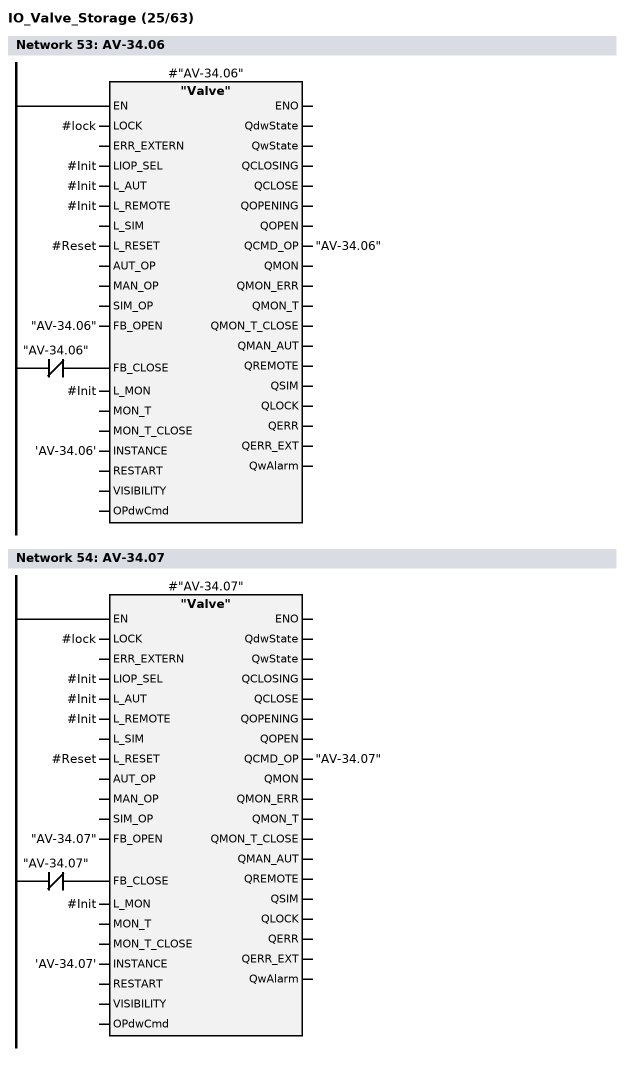
   RUNG wire#powerrail
      #"AV-34.06"(FB_CLOSE := wire#w1, LOCK := #lock, ERR_EXTERN :=, LIOP_SEL := #Init, L_AUT := #Init, L_REMOTE := #Init, L_SIM :=, L_RESET := #Reset, AUT_OP :=, MAN_OP :=, SIM_OP :=, FB_OPEN := "AV-34.06", L_MON := #Init, MON_T :=, MON_T_CLOSE :=, INSTANCE := 'AV-34.06', RESTART :=, VISIBILITY :=, OPdwCmd :=, QdwState =>, QwState =>, QCLOSING =>, QCLOSE =>, QOPENING =>, QOPEN =>, QCMD_OP => "AV-34.06", QMON =>, QMON_ERR =>, QMON_T =>, QMON_T_CLOSE =>, QMAN_AUT =>, QREMOTE =>, QSIM =>, QLOCK =>, QERR =>, QERR_EXT =>, QwAlarm =>)
   END_RUNG
   RUNG wire#powerrail
      I_Contact( "AV-34.06" )
   END_RUNG wire#w1
   // the same network as SCL:
   #"AV-34.06"(LOCK := #lock,   // "Valve"
               LIOP_SEL := #Init,
               L_AUT := #Init,
               L_REMOTE := #Init,
               L_RESET := #Reset,
               FB_OPEN := "AV-34.06",
               FB_CLOSE := NOT "AV-34.06",
               L_MON := #Init,
               INSTANCE := 'AV-34.06',
               QCMD_OP => "AV-34.06");
END_REGION

REGION Network 54: AV-34.07
   RUNG wire#powerrail
      #"AV-34.07"(FB_CLOSE := wire#w1, LOCK := #lock, ERR_EXTERN :=, LIOP_SEL := #Init, L_AUT := #Init, L_REMOTE := #Init, L_SIM :=, L_RESET := #Reset, AUT_OP :=, MAN_OP :=, SIM_OP :=, FB_OPEN := "AV-34.07", L_MON := #Init, MON_T :=, MON_T_CLOSE :=, INSTANCE := 'AV-34.07', RESTART :=, VISIBILITY :=, OPdwCmd :=, QdwState =>, QwState =>, QCLOSING =>, QCLOSE =>, QOPENING =>, QOPEN =>, QCMD_OP => "AV-34.07", QMON =>, QMON_ERR =>, QMON_T =>, QMON_T_CLOSE =>, QMAN_AUT =>, QREMOTE =>, QSIM =>, QLOCK =>, QERR =>, QERR_EXT =>, QwAlarm =>)
   END_RUNG
   RUNG wire#powerrail
      I_Contact( "AV-34.07" )
   END_RUNG wire#w1
   // the same network as SCL:
   #"AV-34.07"(LOCK := #lock,   // "Valve"
               LIOP_SEL := #Init,
               L_AUT := #Init,
               L_REMOTE := #Init,
               L_RESET := #Reset,
               FB_OPEN := "AV-34.07",
               FB_CLOSE := NOT "AV-34.07",
               L_MON := #Init,
               INSTANCE := 'AV-34.07',
               QCMD_OP => "AV-34.07");
END_REGION

REGION Network 55: AV-34.08
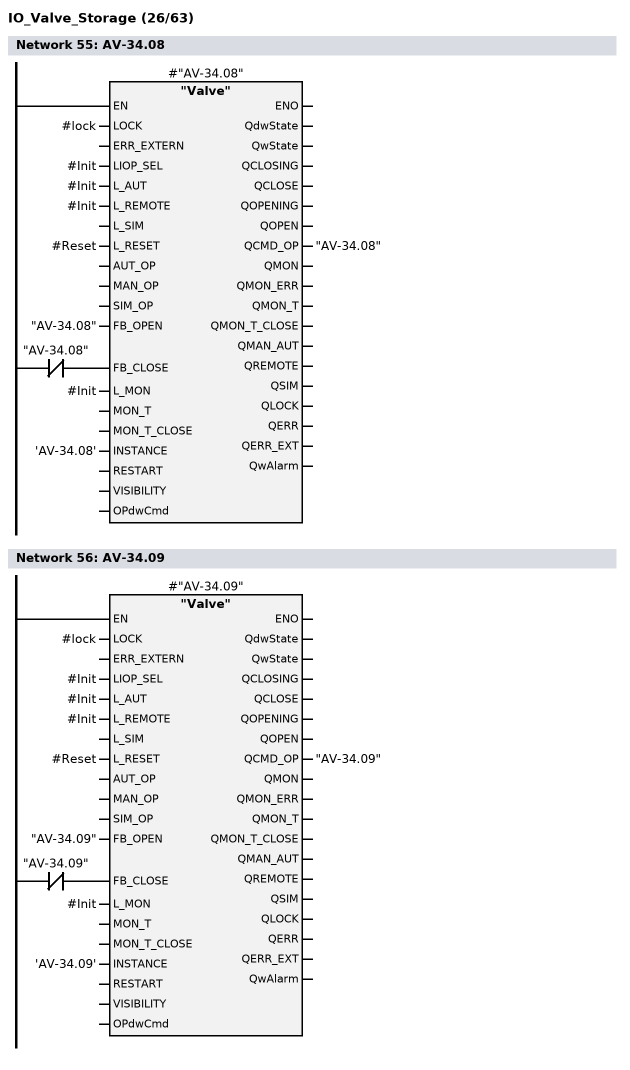
   RUNG wire#powerrail
      #"AV-34.08"(FB_CLOSE := wire#w1, LOCK := #lock, ERR_EXTERN :=, LIOP_SEL := #Init, L_AUT := #Init, L_REMOTE := #Init, L_SIM :=, L_RESET := #Reset, AUT_OP :=, MAN_OP :=, SIM_OP :=, FB_OPEN := "AV-34.08", L_MON := #Init, MON_T :=, MON_T_CLOSE :=, INSTANCE := 'AV-34.08', RESTART :=, VISIBILITY :=, OPdwCmd :=, QdwState =>, QwState =>, QCLOSING =>, QCLOSE =>, QOPENING =>, QOPEN =>, QCMD_OP => "AV-34.08", QMON =>, QMON_ERR =>, QMON_T =>, QMON_T_CLOSE =>, QMAN_AUT =>, QREMOTE =>, QSIM =>, QLOCK =>, QERR =>, QERR_EXT =>, QwAlarm =>)
   END_RUNG
   RUNG wire#powerrail
      I_Contact( "AV-34.08" )
   END_RUNG wire#w1
   // the same network as SCL:
   #"AV-34.08"(LOCK := #lock,   // "Valve"
               LIOP_SEL := #Init,
               L_AUT := #Init,
               L_REMOTE := #Init,
               L_RESET := #Reset,
               FB_OPEN := "AV-34.08",
               FB_CLOSE := NOT "AV-34.08",
               L_MON := #Init,
               INSTANCE := 'AV-34.08',
               QCMD_OP => "AV-34.08");
END_REGION

REGION Network 56: AV-34.09
   RUNG wire#powerrail
      #"AV-34.09"(FB_CLOSE := wire#w1, LOCK := #lock, ERR_EXTERN :=, LIOP_SEL := #Init, L_AUT := #Init, L_REMOTE := #Init, L_SIM :=, L_RESET := #Reset, AUT_OP :=, MAN_OP :=, SIM_OP :=, FB_OPEN := "AV-34.09", L_MON := #Init, MON_T :=, MON_T_CLOSE :=, INSTANCE := 'AV-34.09', RESTART :=, VISIBILITY :=, OPdwCmd :=, QdwState =>, QwState =>, QCLOSING =>, QCLOSE =>, QOPENING =>, QOPEN =>, QCMD_OP => "AV-34.09", QMON =>, QMON_ERR =>, QMON_T =>, QMON_T_CLOSE =>, QMAN_AUT =>, QREMOTE =>, QSIM =>, QLOCK =>, QERR =>, QERR_EXT =>, QwAlarm =>)
   END_RUNG
   RUNG wire#powerrail
      I_Contact( "AV-34.09" )
   END_RUNG wire#w1
   // the same network as SCL:
   #"AV-34.09"(LOCK := #lock,   // "Valve"
               LIOP_SEL := #Init,
               L_AUT := #Init,
               L_REMOTE := #Init,
               L_RESET := #Reset,
               FB_OPEN := "AV-34.09",
               FB_CLOSE := NOT "AV-34.09",
               L_MON := #Init,
               INSTANCE := 'AV-34.09',
               QCMD_OP => "AV-34.09");
END_REGION

REGION Network 57: AV-34.10
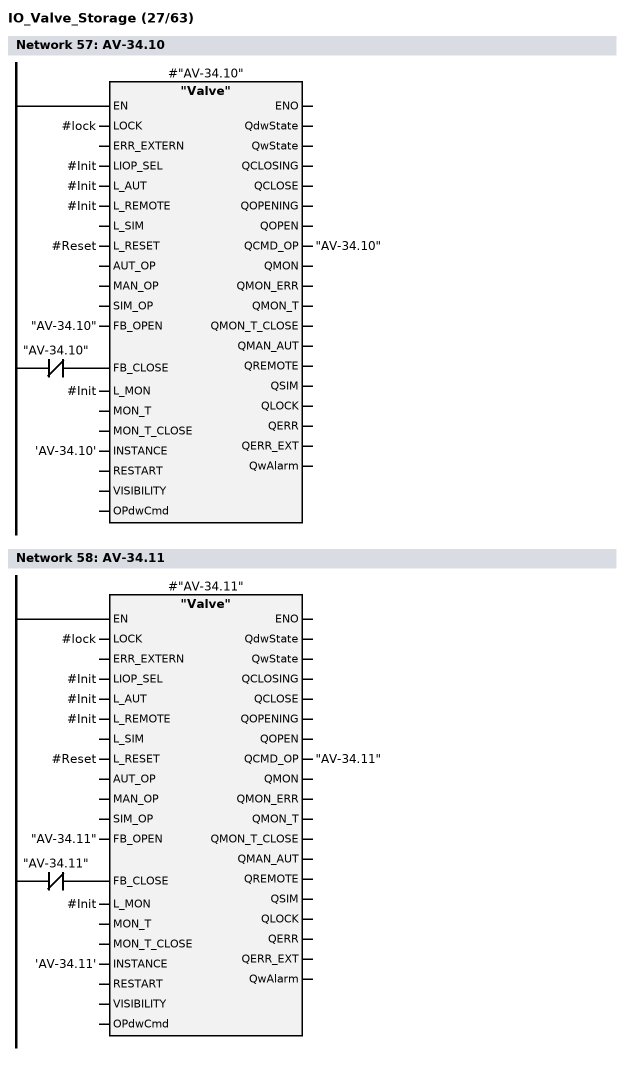
   RUNG wire#powerrail
      #"AV-34.10"(FB_CLOSE := wire#w1, LOCK := #lock, ERR_EXTERN :=, LIOP_SEL := #Init, L_AUT := #Init, L_REMOTE := #Init, L_SIM :=, L_RESET := #Reset, AUT_OP :=, MAN_OP :=, SIM_OP :=, FB_OPEN := "AV-34.10", L_MON := #Init, MON_T :=, MON_T_CLOSE :=, INSTANCE := 'AV-34.10', RESTART :=, VISIBILITY :=, OPdwCmd :=, QdwState =>, QwState =>, QCLOSING =>, QCLOSE =>, QOPENING =>, QOPEN =>, QCMD_OP => "AV-34.10", QMON =>, QMON_ERR =>, QMON_T =>, QMON_T_CLOSE =>, QMAN_AUT =>, QREMOTE =>, QSIM =>, QLOCK =>, QERR =>, QERR_EXT =>, QwAlarm =>)
   END_RUNG
   RUNG wire#powerrail
      I_Contact( "AV-34.10" )
   END_RUNG wire#w1
   // the same network as SCL:
   #"AV-34.10"(LOCK := #lock,   // "Valve"
               LIOP_SEL := #Init,
               L_AUT := #Init,
               L_REMOTE := #Init,
               L_RESET := #Reset,
               FB_OPEN := "AV-34.10",
               FB_CLOSE := NOT "AV-34.10",
               L_MON := #Init,
               INSTANCE := 'AV-34.10',
               QCMD_OP => "AV-34.10");
END_REGION

REGION Network 58: AV-34.11
   RUNG wire#powerrail
      #"AV-34.11"(FB_CLOSE := wire#w1, LOCK := #lock, ERR_EXTERN :=, LIOP_SEL := #Init, L_AUT := #Init, L_REMOTE := #Init, L_SIM :=, L_RESET := #Reset, AUT_OP :=, MAN_OP :=, SIM_OP :=, FB_OPEN := "AV-34.11", L_MON := #Init, MON_T :=, MON_T_CLOSE :=, INSTANCE := 'AV-34.11', RESTART :=, VISIBILITY :=, OPdwCmd :=, QdwState =>, QwState =>, QCLOSING =>, QCLOSE =>, QOPENING =>, QOPEN =>, QCMD_OP => "AV-34.11", QMON =>, QMON_ERR =>, QMON_T =>, QMON_T_CLOSE =>, QMAN_AUT =>, QREMOTE =>, QSIM =>, QLOCK =>, QERR =>, QERR_EXT =>, QwAlarm =>)
   END_RUNG
   RUNG wire#powerrail
      I_Contact( "AV-34.11" )
   END_RUNG wire#w1
   // the same network as SCL:
   #"AV-34.11"(LOCK := #lock,   // "Valve"
               LIOP_SEL := #Init,
               L_AUT := #Init,
               L_REMOTE := #Init,
               L_RESET := #Reset,
               FB_OPEN := "AV-34.11",
               FB_CLOSE := NOT "AV-34.11",
               L_MON := #Init,
               INSTANCE := 'AV-34.11',
               QCMD_OP => "AV-34.11");
END_REGION

REGION Network 59: AV-34.12
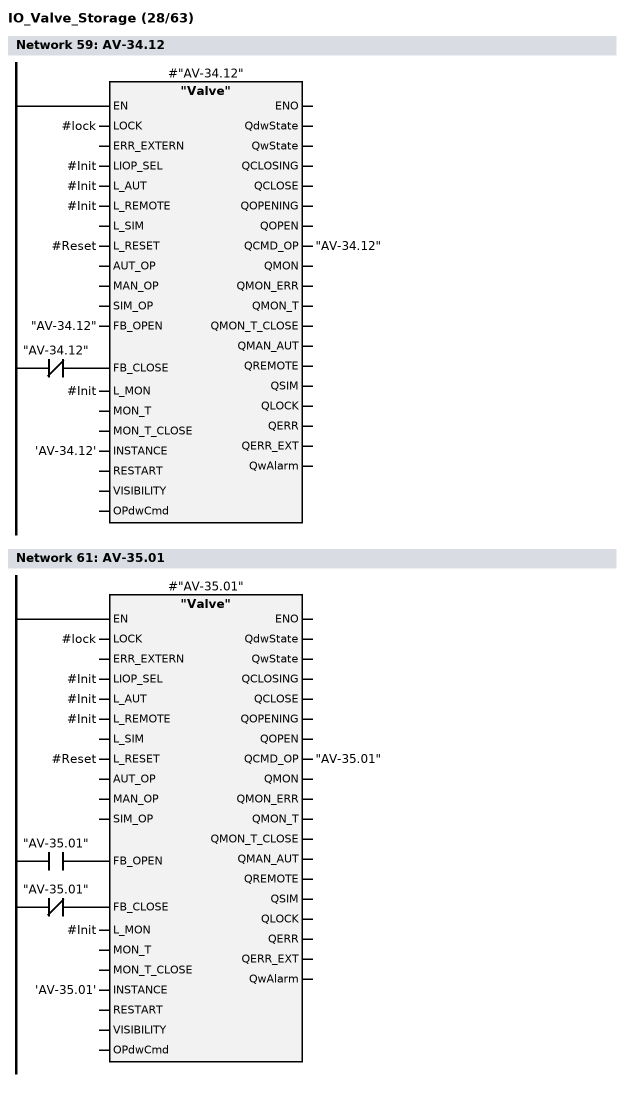
   RUNG wire#powerrail
      #"AV-34.12"(FB_CLOSE := wire#w1, LOCK := #lock, ERR_EXTERN :=, LIOP_SEL := #Init, L_AUT := #Init, L_REMOTE := #Init, L_SIM :=, L_RESET := #Reset, AUT_OP :=, MAN_OP :=, SIM_OP :=, FB_OPEN := "AV-34.12", L_MON := #Init, MON_T :=, MON_T_CLOSE :=, INSTANCE := 'AV-34.12', RESTART :=, VISIBILITY :=, OPdwCmd :=, QdwState =>, QwState =>, QCLOSING =>, QCLOSE =>, QOPENING =>, QOPEN =>, QCMD_OP => "AV-34.12", QMON =>, QMON_ERR =>, QMON_T =>, QMON_T_CLOSE =>, QMAN_AUT =>, QREMOTE =>, QSIM =>, QLOCK =>, QERR =>, QERR_EXT =>, QwAlarm =>)
   END_RUNG
   RUNG wire#powerrail
      I_Contact( "AV-34.12" )
   END_RUNG wire#w1
   // the same network as SCL:
   #"AV-34.12"(LOCK := #lock,   // "Valve"
               LIOP_SEL := #Init,
               L_AUT := #Init,
               L_REMOTE := #Init,
               L_RESET := #Reset,
               FB_OPEN := "AV-34.12",
               FB_CLOSE := NOT "AV-34.12",
               L_MON := #Init,
               INSTANCE := 'AV-34.12',
               QCMD_OP => "AV-34.12");
END_REGION

REGION Network 61: AV-35.01
   RUNG wire#powerrail
      #"AV-35.01"(FB_OPEN := wire#w1, FB_CLOSE := wire#w2, LOCK := #lock, ERR_EXTERN :=, LIOP_SEL := #Init, L_AUT := #Init, L_REMOTE := #Init, L_SIM :=, L_RESET := #Reset, AUT_OP :=, MAN_OP :=, SIM_OP :=, L_MON := #Init, MON_T :=, MON_T_CLOSE :=, INSTANCE := 'AV-35.01', RESTART :=, VISIBILITY :=, OPdwCmd :=, QdwState =>, QwState =>, QCLOSING =>, QCLOSE =>, QOPENING =>, QOPEN =>, QCMD_OP => "AV-35.01", QMON =>, QMON_ERR =>, QMON_T =>, QMON_T_CLOSE =>, QMAN_AUT =>, QREMOTE =>, QSIM =>, QLOCK =>, QERR =>, QERR_EXT =>, QwAlarm =>)
   END_RUNG
   RUNG wire#powerrail
      Contact( "AV-35.01" )
   END_RUNG wire#w1
   RUNG wire#powerrail
      I_Contact( "AV-35.01" )
   END_RUNG wire#w2
   // the same network as SCL:
   #"AV-35.01"(LOCK := #lock,   // "Valve"
               LIOP_SEL := #Init,
               L_AUT := #Init,
               L_REMOTE := #Init,
               L_RESET := #Reset,
               FB_OPEN := "AV-35.01",
               FB_CLOSE := NOT "AV-35.01",
               L_MON := #Init,
               INSTANCE := 'AV-35.01',
               QCMD_OP => "AV-35.01");
END_REGION

REGION Network 62: AV-35.02
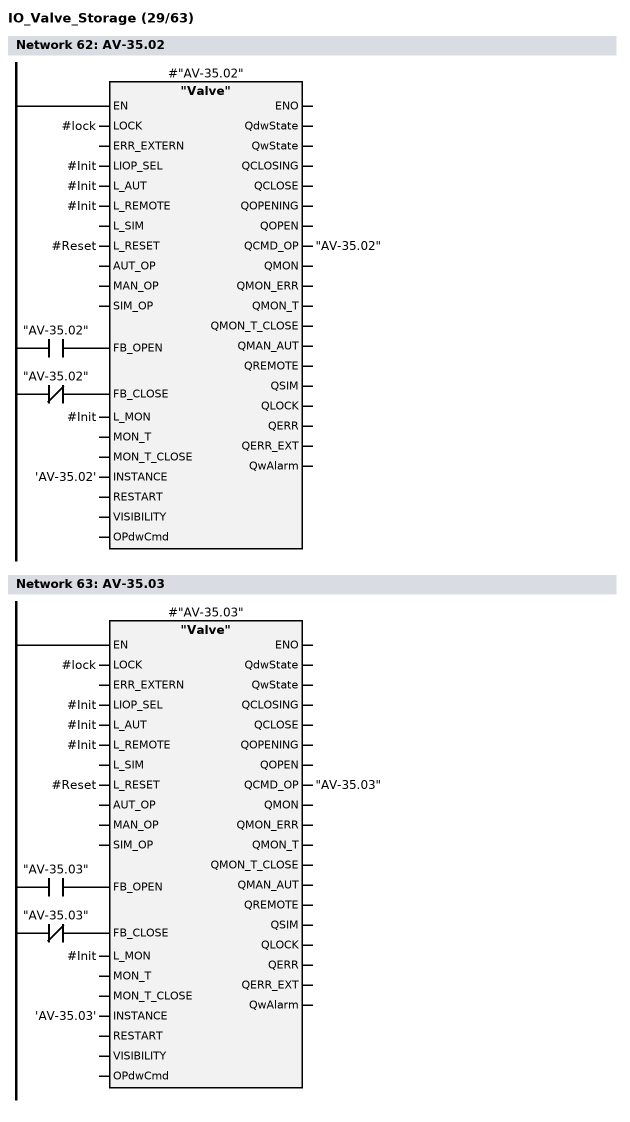
   RUNG wire#powerrail
      #"AV-35.02"(FB_OPEN := wire#w1, FB_CLOSE := wire#w2, LOCK := #lock, ERR_EXTERN :=, LIOP_SEL := #Init, L_AUT := #Init, L_REMOTE := #Init, L_SIM :=, L_RESET := #Reset, AUT_OP :=, MAN_OP :=, SIM_OP :=, L_MON := #Init, MON_T :=, MON_T_CLOSE :=, INSTANCE := 'AV-35.02', RESTART :=, VISIBILITY :=, OPdwCmd :=, QdwState =>, QwState =>, QCLOSING =>, QCLOSE =>, QOPENING =>, QOPEN =>, QCMD_OP => "AV-35.02", QMON =>, QMON_ERR =>, QMON_T =>, QMON_T_CLOSE =>, QMAN_AUT =>, QREMOTE =>, QSIM =>, QLOCK =>, QERR =>, QERR_EXT =>, QwAlarm =>)
   END_RUNG
   RUNG wire#powerrail
      Contact( "AV-35.02" )
   END_RUNG wire#w1
   RUNG wire#powerrail
      I_Contact( "AV-35.02" )
   END_RUNG wire#w2
   // the same network as SCL:
   #"AV-35.02"(LOCK := #lock,   // "Valve"
               LIOP_SEL := #Init,
               L_AUT := #Init,
               L_REMOTE := #Init,
               L_RESET := #Reset,
               FB_OPEN := "AV-35.02",
               FB_CLOSE := NOT "AV-35.02",
               L_MON := #Init,
               INSTANCE := 'AV-35.02',
               QCMD_OP => "AV-35.02");
END_REGION

REGION Network 63: AV-35.03
   RUNG wire#powerrail
      #"AV-35.03"(FB_OPEN := wire#w1, FB_CLOSE := wire#w2, LOCK := #lock, ERR_EXTERN :=, LIOP_SEL := #Init, L_AUT := #Init, L_REMOTE := #Init, L_SIM :=, L_RESET := #Reset, AUT_OP :=, MAN_OP :=, SIM_OP :=, L_MON := #Init, MON_T :=, MON_T_CLOSE :=, INSTANCE := 'AV-35.03', RESTART :=, VISIBILITY :=, OPdwCmd :=, QdwState =>, QwState =>, QCLOSING =>, QCLOSE =>, QOPENING =>, QOPEN =>, QCMD_OP => "AV-35.03", QMON =>, QMON_ERR =>, QMON_T =>, QMON_T_CLOSE =>, QMAN_AUT =>, QREMOTE =>, QSIM =>, QLOCK =>, QERR =>, QERR_EXT =>, QwAlarm =>)
   END_RUNG
   RUNG wire#powerrail
      Contact( "AV-35.03" )
   END_RUNG wire#w1
   RUNG wire#powerrail
      I_Contact( "AV-35.03" )
   END_RUNG wire#w2
   // the same network as SCL:
   #"AV-35.03"(LOCK := #lock,   // "Valve"
               LIOP_SEL := #Init,
               L_AUT := #Init,
               L_REMOTE := #Init,
               L_RESET := #Reset,
               FB_OPEN := "AV-35.03",
               FB_CLOSE := NOT "AV-35.03",
               L_MON := #Init,
               INSTANCE := 'AV-35.03',
               QCMD_OP => "AV-35.03");
END_REGION

REGION Network 64: AV-35.04
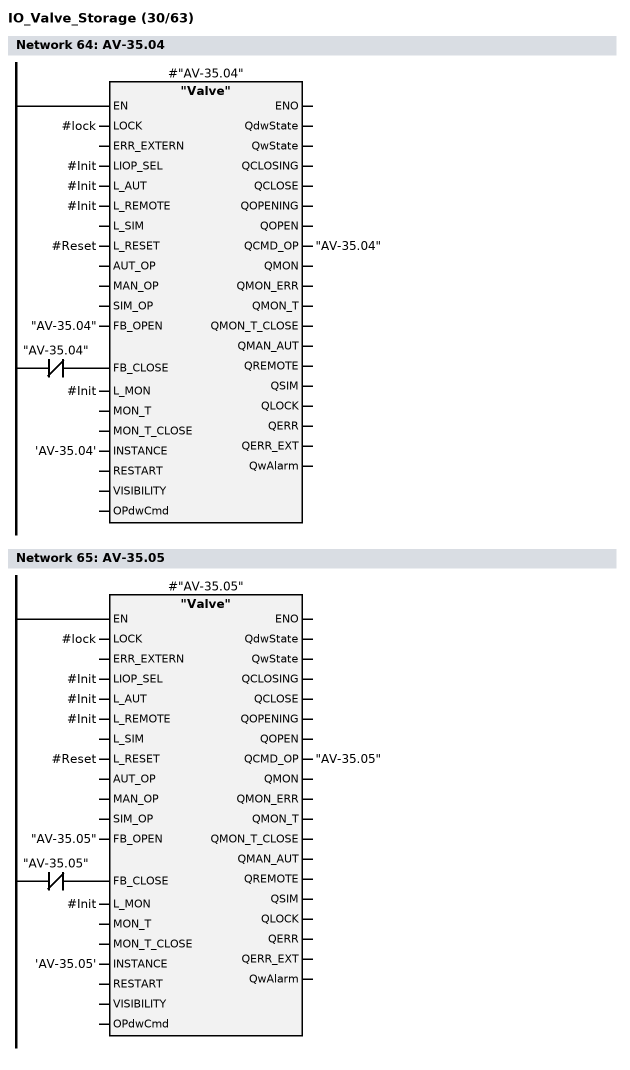
   RUNG wire#powerrail
      #"AV-35.04"(FB_CLOSE := wire#w1, LOCK := #lock, ERR_EXTERN :=, LIOP_SEL := #Init, L_AUT := #Init, L_REMOTE := #Init, L_SIM :=, L_RESET := #Reset, AUT_OP :=, MAN_OP :=, SIM_OP :=, FB_OPEN := "AV-35.04", L_MON := #Init, MON_T :=, MON_T_CLOSE :=, INSTANCE := 'AV-35.04', RESTART :=, VISIBILITY :=, OPdwCmd :=, QdwState =>, QwState =>, QCLOSING =>, QCLOSE =>, QOPENING =>, QOPEN =>, QCMD_OP => "AV-35.04", QMON =>, QMON_ERR =>, QMON_T =>, QMON_T_CLOSE =>, QMAN_AUT =>, QREMOTE =>, QSIM =>, QLOCK =>, QERR =>, QERR_EXT =>, QwAlarm =>)
   END_RUNG
   RUNG wire#powerrail
      I_Contact( "AV-35.04" )
   END_RUNG wire#w1
   // the same network as SCL:
   #"AV-35.04"(LOCK := #lock,   // "Valve"
               LIOP_SEL := #Init,
               L_AUT := #Init,
               L_REMOTE := #Init,
               L_RESET := #Reset,
               FB_OPEN := "AV-35.04",
               FB_CLOSE := NOT "AV-35.04",
               L_MON := #Init,
               INSTANCE := 'AV-35.04',
               QCMD_OP => "AV-35.04");
END_REGION

REGION Network 65: AV-35.05
   RUNG wire#powerrail
      #"AV-35.05"(FB_CLOSE := wire#w1, LOCK := #lock, ERR_EXTERN :=, LIOP_SEL := #Init, L_AUT := #Init, L_REMOTE := #Init, L_SIM :=, L_RESET := #Reset, AUT_OP :=, MAN_OP :=, SIM_OP :=, FB_OPEN := "AV-35.05", L_MON := #Init, MON_T :=, MON_T_CLOSE :=, INSTANCE := 'AV-35.05', RESTART :=, VISIBILITY :=, OPdwCmd :=, QdwState =>, QwState =>, QCLOSING =>, QCLOSE =>, QOPENING =>, QOPEN =>, QCMD_OP => "AV-35.05", QMON =>, QMON_ERR =>, QMON_T =>, QMON_T_CLOSE =>, QMAN_AUT =>, QREMOTE =>, QSIM =>, QLOCK =>, QERR =>, QERR_EXT =>, QwAlarm =>)
   END_RUNG
   RUNG wire#powerrail
      I_Contact( "AV-35.05" )
   END_RUNG wire#w1
   // the same network as SCL:
   #"AV-35.05"(LOCK := #lock,   // "Valve"
               LIOP_SEL := #Init,
               L_AUT := #Init,
               L_REMOTE := #Init,
               L_RESET := #Reset,
               FB_OPEN := "AV-35.05",
               FB_CLOSE := NOT "AV-35.05",
               L_MON := #Init,
               INSTANCE := 'AV-35.05',
               QCMD_OP => "AV-35.05");
END_REGION

REGION Network 66: AV-35.06
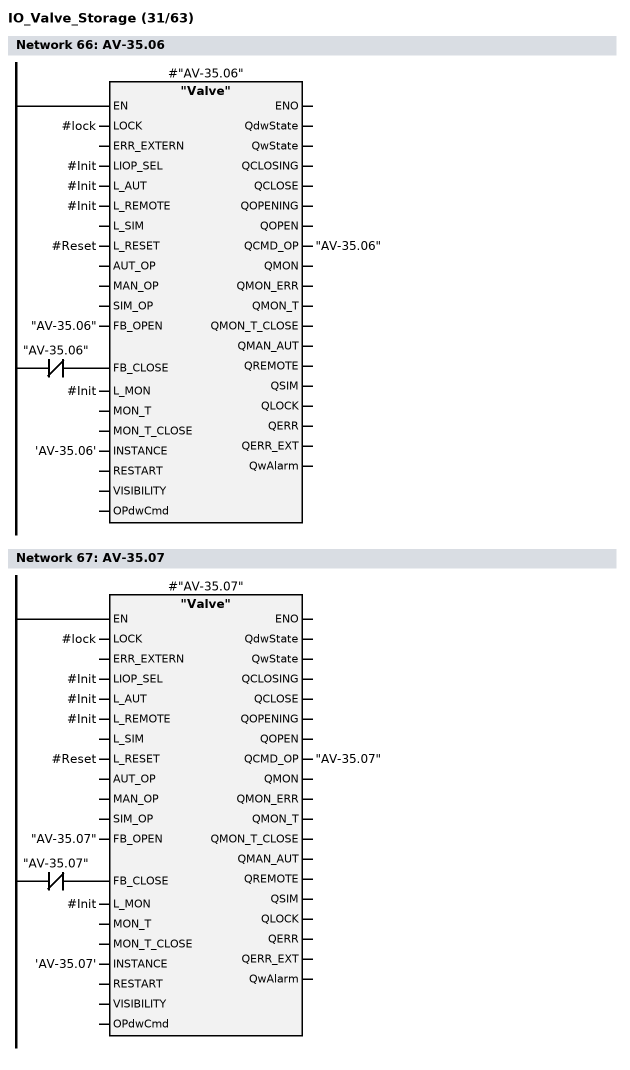
   RUNG wire#powerrail
      #"AV-35.06"(FB_CLOSE := wire#w1, LOCK := #lock, ERR_EXTERN :=, LIOP_SEL := #Init, L_AUT := #Init, L_REMOTE := #Init, L_SIM :=, L_RESET := #Reset, AUT_OP :=, MAN_OP :=, SIM_OP :=, FB_OPEN := "AV-35.06", L_MON := #Init, MON_T :=, MON_T_CLOSE :=, INSTANCE := 'AV-35.06', RESTART :=, VISIBILITY :=, OPdwCmd :=, QdwState =>, QwState =>, QCLOSING =>, QCLOSE =>, QOPENING =>, QOPEN =>, QCMD_OP => "AV-35.06", QMON =>, QMON_ERR =>, QMON_T =>, QMON_T_CLOSE =>, QMAN_AUT =>, QREMOTE =>, QSIM =>, QLOCK =>, QERR =>, QERR_EXT =>, QwAlarm =>)
   END_RUNG
   RUNG wire#powerrail
      I_Contact( "AV-35.06" )
   END_RUNG wire#w1
   // the same network as SCL:
   #"AV-35.06"(LOCK := #lock,   // "Valve"
               LIOP_SEL := #Init,
               L_AUT := #Init,
               L_REMOTE := #Init,
               L_RESET := #Reset,
               FB_OPEN := "AV-35.06",
               FB_CLOSE := NOT "AV-35.06",
               L_MON := #Init,
               INSTANCE := 'AV-35.06',
               QCMD_OP => "AV-35.06");
END_REGION

REGION Network 67: AV-35.07
   RUNG wire#powerrail
      #"AV-35.07"(FB_CLOSE := wire#w1, LOCK := #lock, ERR_EXTERN :=, LIOP_SEL := #Init, L_AUT := #Init, L_REMOTE := #Init, L_SIM :=, L_RESET := #Reset, AUT_OP :=, MAN_OP :=, SIM_OP :=, FB_OPEN := "AV-35.07", L_MON := #Init, MON_T :=, MON_T_CLOSE :=, INSTANCE := 'AV-35.07', RESTART :=, VISIBILITY :=, OPdwCmd :=, QdwState =>, QwState =>, QCLOSING =>, QCLOSE =>, QOPENING =>, QOPEN =>, QCMD_OP => "AV-35.07", QMON =>, QMON_ERR =>, QMON_T =>, QMON_T_CLOSE =>, QMAN_AUT =>, QREMOTE =>, QSIM =>, QLOCK =>, QERR =>, QERR_EXT =>, QwAlarm =>)
   END_RUNG
   RUNG wire#powerrail
      I_Contact( "AV-35.07" )
   END_RUNG wire#w1
   // the same network as SCL:
   #"AV-35.07"(LOCK := #lock,   // "Valve"
               LIOP_SEL := #Init,
               L_AUT := #Init,
               L_REMOTE := #Init,
               L_RESET := #Reset,
               FB_OPEN := "AV-35.07",
               FB_CLOSE := NOT "AV-35.07",
               L_MON := #Init,
               INSTANCE := 'AV-35.07',
               QCMD_OP => "AV-35.07");
END_REGION

REGION Network 68: AV-35.08
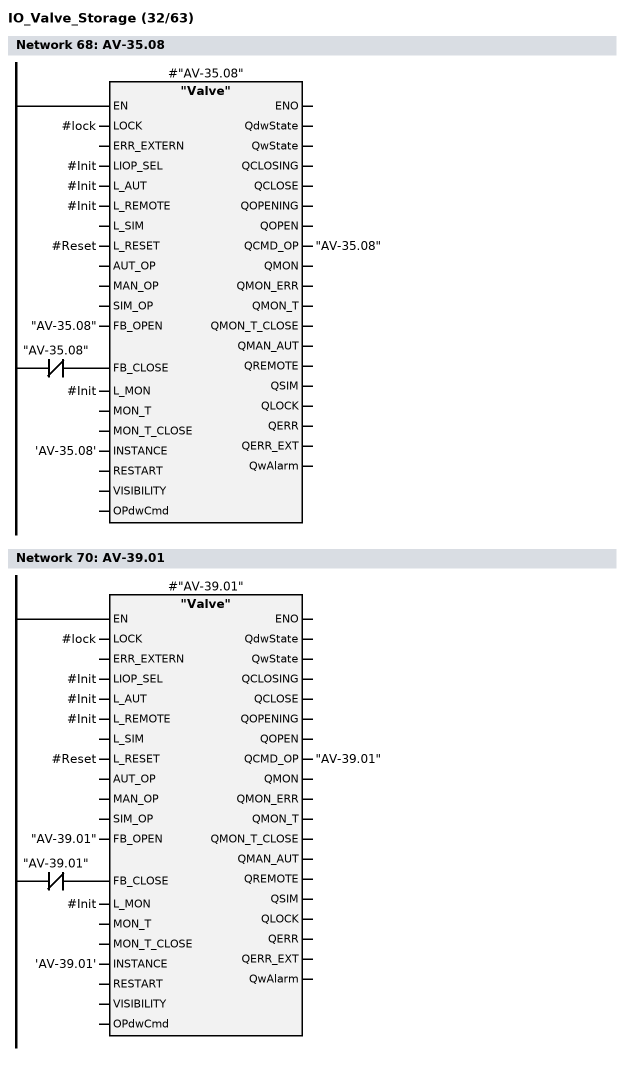
   RUNG wire#powerrail
      #"AV-35.08"(FB_CLOSE := wire#w1, LOCK := #lock, ERR_EXTERN :=, LIOP_SEL := #Init, L_AUT := #Init, L_REMOTE := #Init, L_SIM :=, L_RESET := #Reset, AUT_OP :=, MAN_OP :=, SIM_OP :=, FB_OPEN := "AV-35.08", L_MON := #Init, MON_T :=, MON_T_CLOSE :=, INSTANCE := 'AV-35.08', RESTART :=, VISIBILITY :=, OPdwCmd :=, QdwState =>, QwState =>, QCLOSING =>, QCLOSE =>, QOPENING =>, QOPEN =>, QCMD_OP => "AV-35.08", QMON =>, QMON_ERR =>, QMON_T =>, QMON_T_CLOSE =>, QMAN_AUT =>, QREMOTE =>, QSIM =>, QLOCK =>, QERR =>, QERR_EXT =>, QwAlarm =>)
   END_RUNG
   RUNG wire#powerrail
      I_Contact( "AV-35.08" )
   END_RUNG wire#w1
   // the same network as SCL:
   #"AV-35.08"(LOCK := #lock,   // "Valve"
               LIOP_SEL := #Init,
               L_AUT := #Init,
               L_REMOTE := #Init,
               L_RESET := #Reset,
               FB_OPEN := "AV-35.08",
               FB_CLOSE := NOT "AV-35.08",
               L_MON := #Init,
               INSTANCE := 'AV-35.08',
               QCMD_OP => "AV-35.08");
END_REGION

REGION Network 70: AV-39.01
   RUNG wire#powerrail
      #"AV-39.01"(FB_CLOSE := wire#w1, LOCK := #lock, ERR_EXTERN :=, LIOP_SEL := #Init, L_AUT := #Init, L_REMOTE := #Init, L_SIM :=, L_RESET := #Reset, AUT_OP :=, MAN_OP :=, SIM_OP :=, FB_OPEN := "AV-39.01", L_MON := #Init, MON_T :=, MON_T_CLOSE :=, INSTANCE := 'AV-39.01', RESTART :=, VISIBILITY :=, OPdwCmd :=, QdwState =>, QwState =>, QCLOSING =>, QCLOSE =>, QOPENING =>, QOPEN =>, QCMD_OP => "AV-39.01", QMON =>, QMON_ERR =>, QMON_T =>, QMON_T_CLOSE =>, QMAN_AUT =>, QREMOTE =>, QSIM =>, QLOCK =>, QERR =>, QERR_EXT =>, QwAlarm =>)
   END_RUNG
   RUNG wire#powerrail
      I_Contact( "AV-39.01" )
   END_RUNG wire#w1
   // the same network as SCL:
   #"AV-39.01"(LOCK := #lock,   // "Valve"
               LIOP_SEL := #Init,
               L_AUT := #Init,
               L_REMOTE := #Init,
               L_RESET := #Reset,
               FB_OPEN := "AV-39.01",
               FB_CLOSE := NOT "AV-39.01",
               L_MON := #Init,
               INSTANCE := 'AV-39.01',
               QCMD_OP => "AV-39.01");
END_REGION

REGION Network 71: AV-39.02
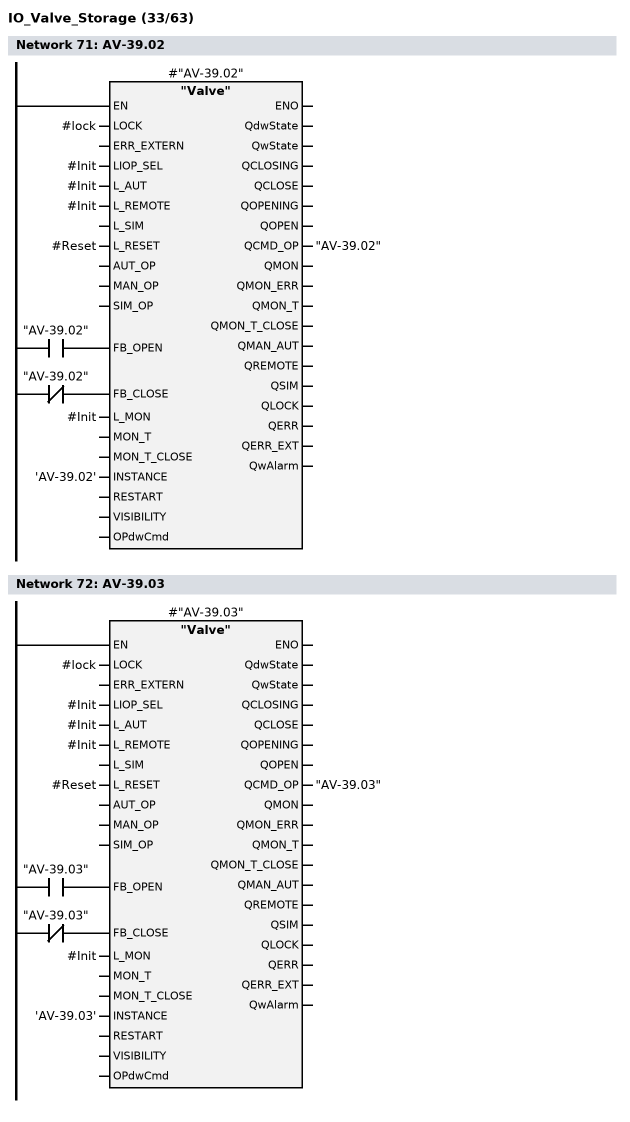
   RUNG wire#powerrail
      #"AV-39.02"(FB_OPEN := wire#w1, FB_CLOSE := wire#w2, LOCK := #lock, ERR_EXTERN :=, LIOP_SEL := #Init, L_AUT := #Init, L_REMOTE := #Init, L_SIM :=, L_RESET := #Reset, AUT_OP :=, MAN_OP :=, SIM_OP :=, L_MON := #Init, MON_T :=, MON_T_CLOSE :=, INSTANCE := 'AV-39.02', RESTART :=, VISIBILITY :=, OPdwCmd :=, QdwState =>, QwState =>, QCLOSING =>, QCLOSE =>, QOPENING =>, QOPEN =>, QCMD_OP => "AV-39.02", QMON =>, QMON_ERR =>, QMON_T =>, QMON_T_CLOSE =>, QMAN_AUT =>, QREMOTE =>, QSIM =>, QLOCK =>, QERR =>, QERR_EXT =>, QwAlarm =>)
   END_RUNG
   RUNG wire#powerrail
      Contact( "AV-39.02" )
   END_RUNG wire#w1
   RUNG wire#powerrail
      I_Contact( "AV-39.02" )
   END_RUNG wire#w2
   // the same network as SCL:
   #"AV-39.02"(LOCK := #lock,   // "Valve"
               LIOP_SEL := #Init,
               L_AUT := #Init,
               L_REMOTE := #Init,
               L_RESET := #Reset,
               FB_OPEN := "AV-39.02",
               FB_CLOSE := NOT "AV-39.02",
               L_MON := #Init,
               INSTANCE := 'AV-39.02',
               QCMD_OP => "AV-39.02");
END_REGION

REGION Network 72: AV-39.03
   RUNG wire#powerrail
      #"AV-39.03"(FB_OPEN := wire#w1, FB_CLOSE := wire#w2, LOCK := #lock, ERR_EXTERN :=, LIOP_SEL := #Init, L_AUT := #Init, L_REMOTE := #Init, L_SIM :=, L_RESET := #Reset, AUT_OP :=, MAN_OP :=, SIM_OP :=, L_MON := #Init, MON_T :=, MON_T_CLOSE :=, INSTANCE := 'AV-39.03', RESTART :=, VISIBILITY :=, OPdwCmd :=, QdwState =>, QwState =>, QCLOSING =>, QCLOSE =>, QOPENING =>, QOPEN =>, QCMD_OP => "AV-39.03", QMON =>, QMON_ERR =>, QMON_T =>, QMON_T_CLOSE =>, QMAN_AUT =>, QREMOTE =>, QSIM =>, QLOCK =>, QERR =>, QERR_EXT =>, QwAlarm =>)
   END_RUNG
   RUNG wire#powerrail
      Contact( "AV-39.03" )
   END_RUNG wire#w1
   RUNG wire#powerrail
      I_Contact( "AV-39.03" )
   END_RUNG wire#w2
   // the same network as SCL:
   #"AV-39.03"(LOCK := #lock,   // "Valve"
               LIOP_SEL := #Init,
               L_AUT := #Init,
               L_REMOTE := #Init,
               L_RESET := #Reset,
               FB_OPEN := "AV-39.03",
               FB_CLOSE := NOT "AV-39.03",
               L_MON := #Init,
               INSTANCE := 'AV-39.03',
               QCMD_OP => "AV-39.03");
END_REGION

REGION Network 73: AV-39.04
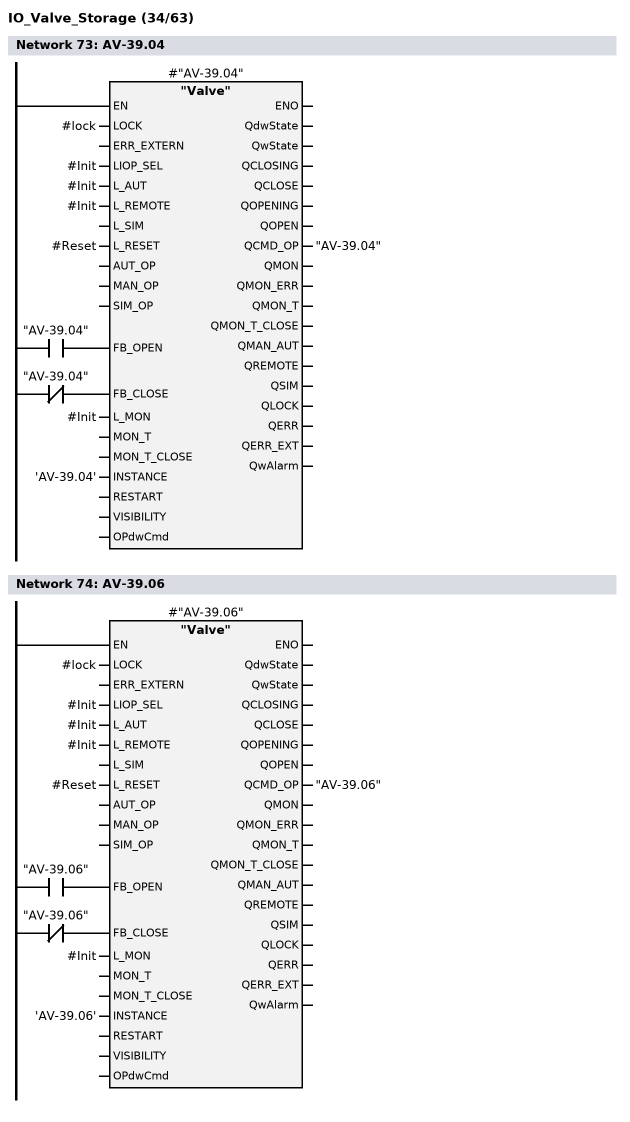
   RUNG wire#powerrail
      #"AV-39.04"(FB_OPEN := wire#w1, FB_CLOSE := wire#w2, LOCK := #lock, ERR_EXTERN :=, LIOP_SEL := #Init, L_AUT := #Init, L_REMOTE := #Init, L_SIM :=, L_RESET := #Reset, AUT_OP :=, MAN_OP :=, SIM_OP :=, L_MON := #Init, MON_T :=, MON_T_CLOSE :=, INSTANCE := 'AV-39.04', RESTART :=, VISIBILITY :=, OPdwCmd :=, QdwState =>, QwState =>, QCLOSING =>, QCLOSE =>, QOPENING =>, QOPEN =>, QCMD_OP => "AV-39.04", QMON =>, QMON_ERR =>, QMON_T =>, QMON_T_CLOSE =>, QMAN_AUT =>, QREMOTE =>, QSIM =>, QLOCK =>, QERR =>, QERR_EXT =>, QwAlarm =>)
   END_RUNG
   RUNG wire#powerrail
      Contact( "AV-39.04" )
   END_RUNG wire#w1
   RUNG wire#powerrail
      I_Contact( "AV-39.04" )
   END_RUNG wire#w2
   // the same network as SCL:
   #"AV-39.04"(LOCK := #lock,   // "Valve"
               LIOP_SEL := #Init,
               L_AUT := #Init,
               L_REMOTE := #Init,
               L_RESET := #Reset,
               FB_OPEN := "AV-39.04",
               FB_CLOSE := NOT "AV-39.04",
               L_MON := #Init,
               INSTANCE := 'AV-39.04',
               QCMD_OP => "AV-39.04");
END_REGION

REGION Network 74: AV-39.06
   RUNG wire#powerrail
      #"AV-39.06"(FB_OPEN := wire#w1, FB_CLOSE := wire#w2, LOCK := #lock, ERR_EXTERN :=, LIOP_SEL := #Init, L_AUT := #Init, L_REMOTE := #Init, L_SIM :=, L_RESET := #Reset, AUT_OP :=, MAN_OP :=, SIM_OP :=, L_MON := #Init, MON_T :=, MON_T_CLOSE :=, INSTANCE := 'AV-39.06', RESTART :=, VISIBILITY :=, OPdwCmd :=, QdwState =>, QwState =>, QCLOSING =>, QCLOSE =>, QOPENING =>, QOPEN =>, QCMD_OP => "AV-39.06", QMON =>, QMON_ERR =>, QMON_T =>, QMON_T_CLOSE =>, QMAN_AUT =>, QREMOTE =>, QSIM =>, QLOCK =>, QERR =>, QERR_EXT =>, QwAlarm =>)
   END_RUNG
   RUNG wire#powerrail
      Contact( "AV-39.06" )
   END_RUNG wire#w1
   RUNG wire#powerrail
      I_Contact( "AV-39.06" )
   END_RUNG wire#w2
   // the same network as SCL:
   #"AV-39.06"(LOCK := #lock,   // "Valve"
               LIOP_SEL := #Init,
               L_AUT := #Init,
               L_REMOTE := #Init,
               L_RESET := #Reset,
               FB_OPEN := "AV-39.06",
               FB_CLOSE := NOT "AV-39.06",
               L_MON := #Init,
               INSTANCE := 'AV-39.06',
               QCMD_OP => "AV-39.06");
END_REGION

REGION Network 76: AV-79.01
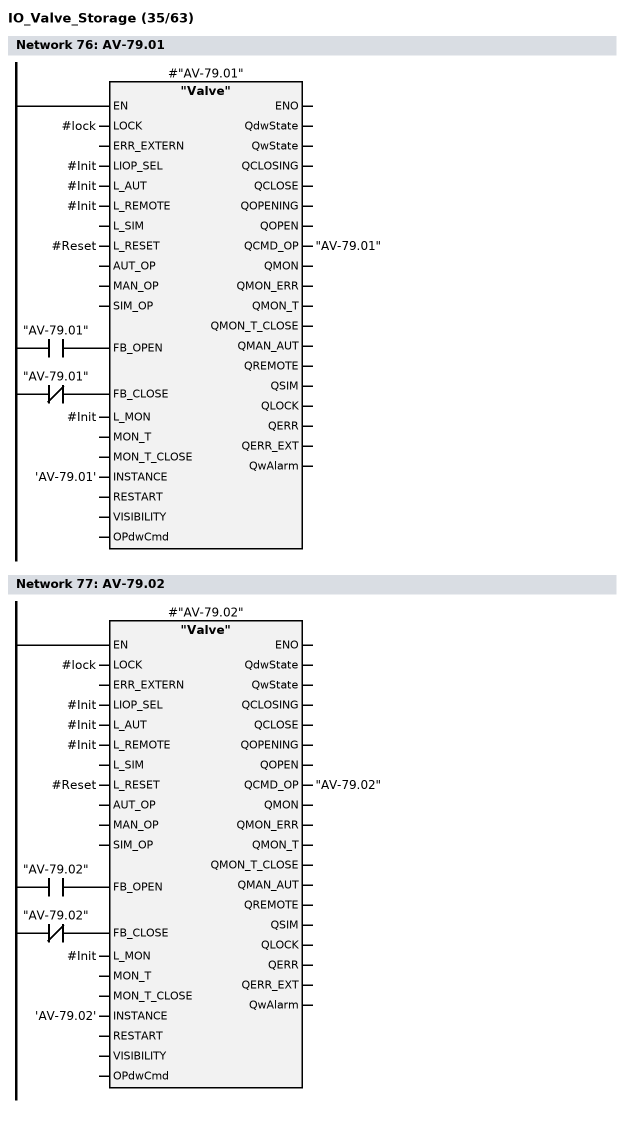
   RUNG wire#powerrail
      #"AV-79.01"(FB_OPEN := wire#w1, FB_CLOSE := wire#w2, LOCK := #lock, ERR_EXTERN :=, LIOP_SEL := #Init, L_AUT := #Init, L_REMOTE := #Init, L_SIM :=, L_RESET := #Reset, AUT_OP :=, MAN_OP :=, SIM_OP :=, L_MON := #Init, MON_T :=, MON_T_CLOSE :=, INSTANCE := 'AV-79.01', RESTART :=, VISIBILITY :=, OPdwCmd :=, QdwState =>, QwState =>, QCLOSING =>, QCLOSE =>, QOPENING =>, QOPEN =>, QCMD_OP => "AV-79.01", QMON =>, QMON_ERR =>, QMON_T =>, QMON_T_CLOSE =>, QMAN_AUT =>, QREMOTE =>, QSIM =>, QLOCK =>, QERR =>, QERR_EXT =>, QwAlarm =>)
   END_RUNG
   RUNG wire#powerrail
      Contact( "AV-79.01" )
   END_RUNG wire#w1
   RUNG wire#powerrail
      I_Contact( "AV-79.01" )
   END_RUNG wire#w2
   // the same network as SCL:
   #"AV-79.01"(LOCK := #lock,   // "Valve"
               LIOP_SEL := #Init,
               L_AUT := #Init,
               L_REMOTE := #Init,
               L_RESET := #Reset,
               FB_OPEN := "AV-79.01",
               FB_CLOSE := NOT "AV-79.01",
               L_MON := #Init,
               INSTANCE := 'AV-79.01',
               QCMD_OP => "AV-79.01");
END_REGION

REGION Network 77: AV-79.02
   RUNG wire#powerrail
      #"AV-79.02"(FB_OPEN := wire#w1, FB_CLOSE := wire#w2, LOCK := #lock, ERR_EXTERN :=, LIOP_SEL := #Init, L_AUT := #Init, L_REMOTE := #Init, L_SIM :=, L_RESET := #Reset, AUT_OP :=, MAN_OP :=, SIM_OP :=, L_MON := #Init, MON_T :=, MON_T_CLOSE :=, INSTANCE := 'AV-79.02', RESTART :=, VISIBILITY :=, OPdwCmd :=, QdwState =>, QwState =>, QCLOSING =>, QCLOSE =>, QOPENING =>, QOPEN =>, QCMD_OP => "AV-79.02", QMON =>, QMON_ERR =>, QMON_T =>, QMON_T_CLOSE =>, QMAN_AUT =>, QREMOTE =>, QSIM =>, QLOCK =>, QERR =>, QERR_EXT =>, QwAlarm =>)
   END_RUNG
   RUNG wire#powerrail
      Contact( "AV-79.02" )
   END_RUNG wire#w1
   RUNG wire#powerrail
      I_Contact( "AV-79.02" )
   END_RUNG wire#w2
   // the same network as SCL:
   #"AV-79.02"(LOCK := #lock,   // "Valve"
               LIOP_SEL := #Init,
               L_AUT := #Init,
               L_REMOTE := #Init,
               L_RESET := #Reset,
               FB_OPEN := "AV-79.02",
               FB_CLOSE := NOT "AV-79.02",
               L_MON := #Init,
               INSTANCE := 'AV-79.02',
               QCMD_OP => "AV-79.02");
END_REGION

REGION Network 78: AV-79.03
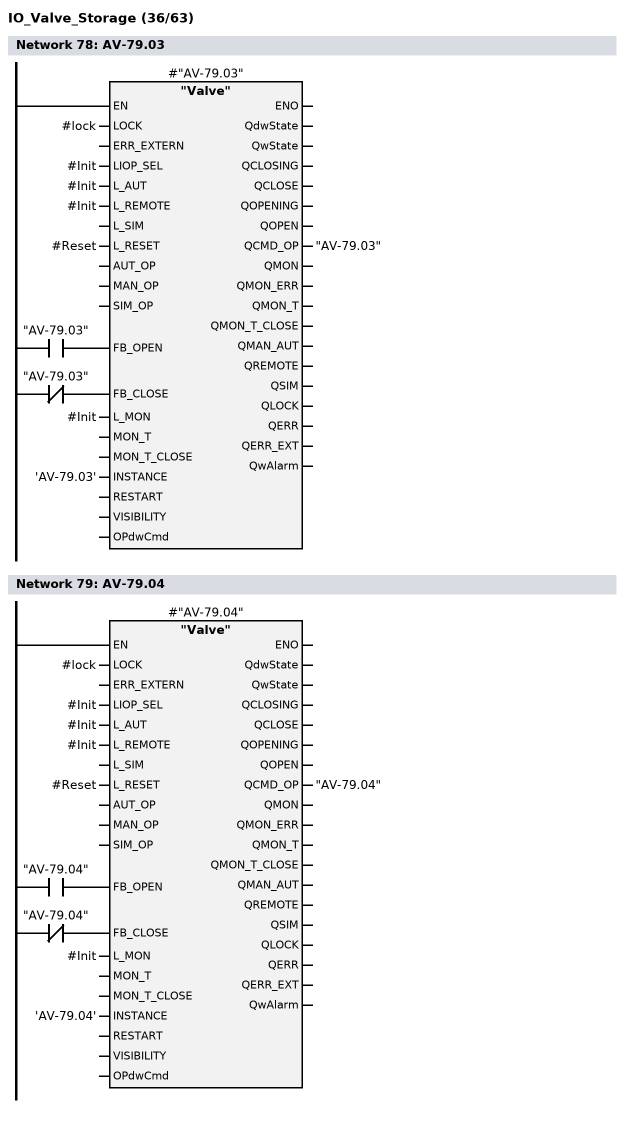
   RUNG wire#powerrail
      #"AV-79.03"(FB_OPEN := wire#w1, FB_CLOSE := wire#w2, LOCK := #lock, ERR_EXTERN :=, LIOP_SEL := #Init, L_AUT := #Init, L_REMOTE := #Init, L_SIM :=, L_RESET := #Reset, AUT_OP :=, MAN_OP :=, SIM_OP :=, L_MON := #Init, MON_T :=, MON_T_CLOSE :=, INSTANCE := 'AV-79.03', RESTART :=, VISIBILITY :=, OPdwCmd :=, QdwState =>, QwState =>, QCLOSING =>, QCLOSE =>, QOPENING =>, QOPEN =>, QCMD_OP => "AV-79.03", QMON =>, QMON_ERR =>, QMON_T =>, QMON_T_CLOSE =>, QMAN_AUT =>, QREMOTE =>, QSIM =>, QLOCK =>, QERR =>, QERR_EXT =>, QwAlarm =>)
   END_RUNG
   RUNG wire#powerrail
      Contact( "AV-79.03" )
   END_RUNG wire#w1
   RUNG wire#powerrail
      I_Contact( "AV-79.03" )
   END_RUNG wire#w2
   // the same network as SCL:
   #"AV-79.03"(LOCK := #lock,   // "Valve"
               LIOP_SEL := #Init,
               L_AUT := #Init,
               L_REMOTE := #Init,
               L_RESET := #Reset,
               FB_OPEN := "AV-79.03",
               FB_CLOSE := NOT "AV-79.03",
               L_MON := #Init,
               INSTANCE := 'AV-79.03',
               QCMD_OP => "AV-79.03");
END_REGION

REGION Network 79: AV-79.04
   RUNG wire#powerrail
      #"AV-79.04"(FB_OPEN := wire#w1, FB_CLOSE := wire#w2, LOCK := #lock, ERR_EXTERN :=, LIOP_SEL := #Init, L_AUT := #Init, L_REMOTE := #Init, L_SIM :=, L_RESET := #Reset, AUT_OP :=, MAN_OP :=, SIM_OP :=, L_MON := #Init, MON_T :=, MON_T_CLOSE :=, INSTANCE := 'AV-79.04', RESTART :=, VISIBILITY :=, OPdwCmd :=, QdwState =>, QwState =>, QCLOSING =>, QCLOSE =>, QOPENING =>, QOPEN =>, QCMD_OP => "AV-79.04", QMON =>, QMON_ERR =>, QMON_T =>, QMON_T_CLOSE =>, QMAN_AUT =>, QREMOTE =>, QSIM =>, QLOCK =>, QERR =>, QERR_EXT =>, QwAlarm =>)
   END_RUNG
   RUNG wire#powerrail
      Contact( "AV-79.04" )
   END_RUNG wire#w1
   RUNG wire#powerrail
      I_Contact( "AV-79.04" )
   END_RUNG wire#w2
   // the same network as SCL:
   #"AV-79.04"(LOCK := #lock,   // "Valve"
               LIOP_SEL := #Init,
               L_AUT := #Init,
               L_REMOTE := #Init,
               L_RESET := #Reset,
               FB_OPEN := "AV-79.04",
               FB_CLOSE := NOT "AV-79.04",
               L_MON := #Init,
               INSTANCE := 'AV-79.04',
               QCMD_OP => "AV-79.04");
END_REGION

REGION Network 80: AV-79.05
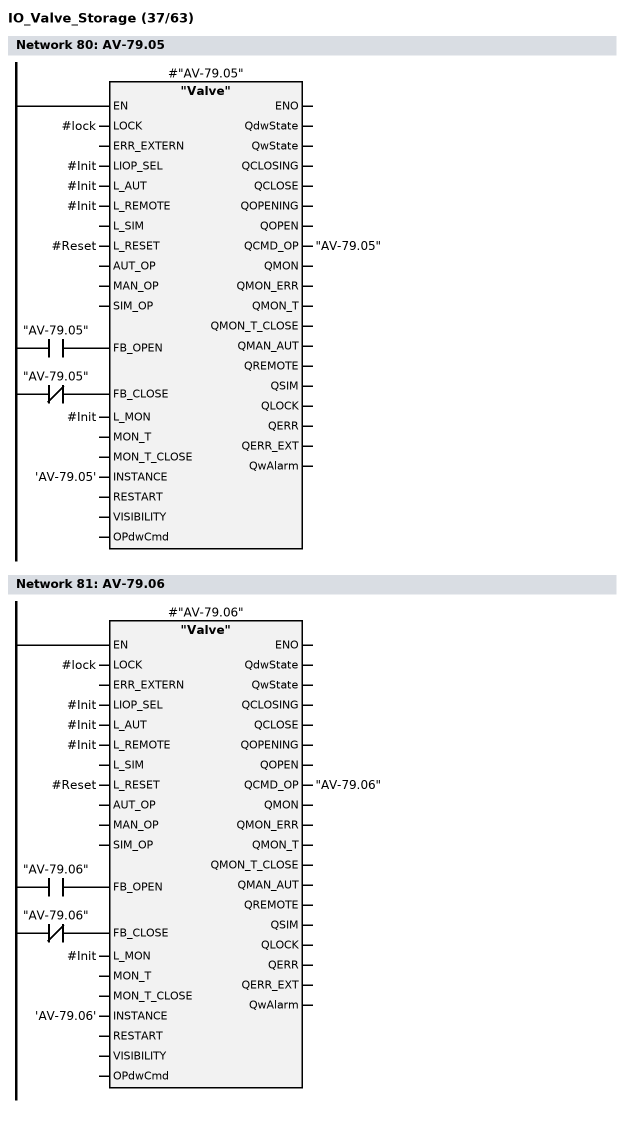
   RUNG wire#powerrail
      #"AV-79.05"(FB_OPEN := wire#w1, FB_CLOSE := wire#w2, LOCK := #lock, ERR_EXTERN :=, LIOP_SEL := #Init, L_AUT := #Init, L_REMOTE := #Init, L_SIM :=, L_RESET := #Reset, AUT_OP :=, MAN_OP :=, SIM_OP :=, L_MON := #Init, MON_T :=, MON_T_CLOSE :=, INSTANCE := 'AV-79.05', RESTART :=, VISIBILITY :=, OPdwCmd :=, QdwState =>, QwState =>, QCLOSING =>, QCLOSE =>, QOPENING =>, QOPEN =>, QCMD_OP => "AV-79.05", QMON =>, QMON_ERR =>, QMON_T =>, QMON_T_CLOSE =>, QMAN_AUT =>, QREMOTE =>, QSIM =>, QLOCK =>, QERR =>, QERR_EXT =>, QwAlarm =>)
   END_RUNG
   RUNG wire#powerrail
      Contact( "AV-79.05" )
   END_RUNG wire#w1
   RUNG wire#powerrail
      I_Contact( "AV-79.05" )
   END_RUNG wire#w2
   // the same network as SCL:
   #"AV-79.05"(LOCK := #lock,   // "Valve"
               LIOP_SEL := #Init,
               L_AUT := #Init,
               L_REMOTE := #Init,
               L_RESET := #Reset,
               FB_OPEN := "AV-79.05",
               FB_CLOSE := NOT "AV-79.05",
               L_MON := #Init,
               INSTANCE := 'AV-79.05',
               QCMD_OP => "AV-79.05");
END_REGION

REGION Network 81: AV-79.06
   RUNG wire#powerrail
      #"AV-79.06"(FB_OPEN := wire#w1, FB_CLOSE := wire#w2, LOCK := #lock, ERR_EXTERN :=, LIOP_SEL := #Init, L_AUT := #Init, L_REMOTE := #Init, L_SIM :=, L_RESET := #Reset, AUT_OP :=, MAN_OP :=, SIM_OP :=, L_MON := #Init, MON_T :=, MON_T_CLOSE :=, INSTANCE := 'AV-79.06', RESTART :=, VISIBILITY :=, OPdwCmd :=, QdwState =>, QwState =>, QCLOSING =>, QCLOSE =>, QOPENING =>, QOPEN =>, QCMD_OP => "AV-79.06", QMON =>, QMON_ERR =>, QMON_T =>, QMON_T_CLOSE =>, QMAN_AUT =>, QREMOTE =>, QSIM =>, QLOCK =>, QERR =>, QERR_EXT =>, QwAlarm =>)
   END_RUNG
   RUNG wire#powerrail
      Contact( "AV-79.06" )
   END_RUNG wire#w1
   RUNG wire#powerrail
      I_Contact( "AV-79.06" )
   END_RUNG wire#w2
   // the same network as SCL:
   #"AV-79.06"(LOCK := #lock,   // "Valve"
               LIOP_SEL := #Init,
               L_AUT := #Init,
               L_REMOTE := #Init,
               L_RESET := #Reset,
               FB_OPEN := "AV-79.06",
               FB_CLOSE := NOT "AV-79.06",
               L_MON := #Init,
               INSTANCE := 'AV-79.06',
               QCMD_OP => "AV-79.06");
END_REGION

REGION Network 82: AV-79.07
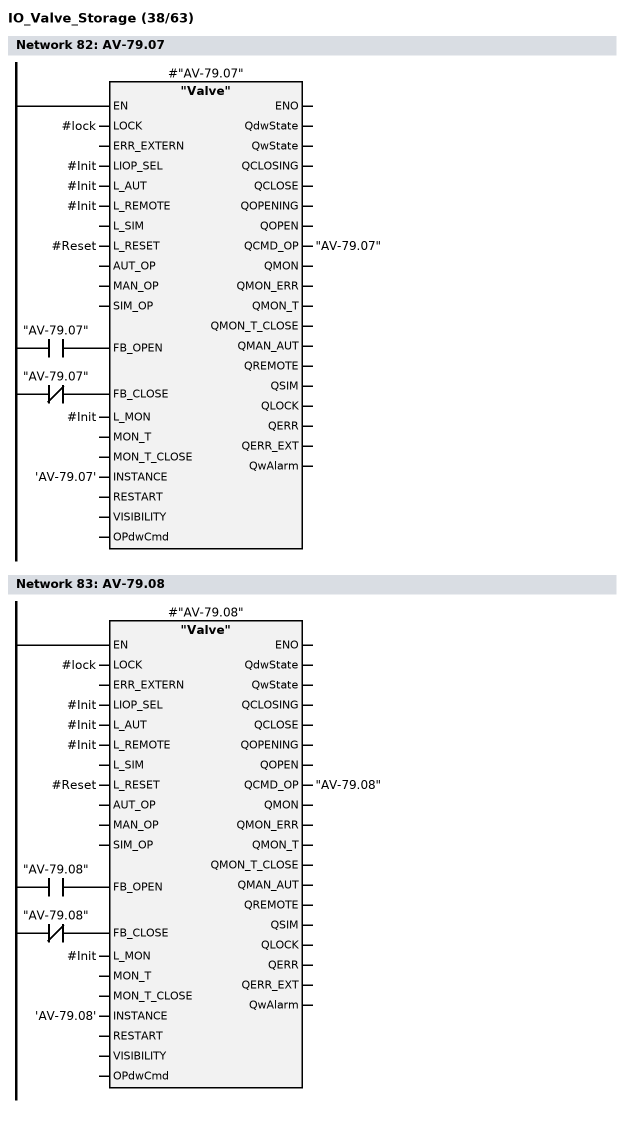
   RUNG wire#powerrail
      #"AV-79.07"(FB_OPEN := wire#w1, FB_CLOSE := wire#w2, LOCK := #lock, ERR_EXTERN :=, LIOP_SEL := #Init, L_AUT := #Init, L_REMOTE := #Init, L_SIM :=, L_RESET := #Reset, AUT_OP :=, MAN_OP :=, SIM_OP :=, L_MON := #Init, MON_T :=, MON_T_CLOSE :=, INSTANCE := 'AV-79.07', RESTART :=, VISIBILITY :=, OPdwCmd :=, QdwState =>, QwState =>, QCLOSING =>, QCLOSE =>, QOPENING =>, QOPEN =>, QCMD_OP => "AV-79.07", QMON =>, QMON_ERR =>, QMON_T =>, QMON_T_CLOSE =>, QMAN_AUT =>, QREMOTE =>, QSIM =>, QLOCK =>, QERR =>, QERR_EXT =>, QwAlarm =>)
   END_RUNG
   RUNG wire#powerrail
      Contact( "AV-79.07" )
   END_RUNG wire#w1
   RUNG wire#powerrail
      I_Contact( "AV-79.07" )
   END_RUNG wire#w2
   // the same network as SCL:
   #"AV-79.07"(LOCK := #lock,   // "Valve"
               LIOP_SEL := #Init,
               L_AUT := #Init,
               L_REMOTE := #Init,
               L_RESET := #Reset,
               FB_OPEN := "AV-79.07",
               FB_CLOSE := NOT "AV-79.07",
               L_MON := #Init,
               INSTANCE := 'AV-79.07',
               QCMD_OP => "AV-79.07");
END_REGION

REGION Network 83: AV-79.08
   RUNG wire#powerrail
      #"AV-79.08"(FB_OPEN := wire#w1, FB_CLOSE := wire#w2, LOCK := #lock, ERR_EXTERN :=, LIOP_SEL := #Init, L_AUT := #Init, L_REMOTE := #Init, L_SIM :=, L_RESET := #Reset, AUT_OP :=, MAN_OP :=, SIM_OP :=, L_MON := #Init, MON_T :=, MON_T_CLOSE :=, INSTANCE := 'AV-79.08', RESTART :=, VISIBILITY :=, OPdwCmd :=, QdwState =>, QwState =>, QCLOSING =>, QCLOSE =>, QOPENING =>, QOPEN =>, QCMD_OP => "AV-79.08", QMON =>, QMON_ERR =>, QMON_T =>, QMON_T_CLOSE =>, QMAN_AUT =>, QREMOTE =>, QSIM =>, QLOCK =>, QERR =>, QERR_EXT =>, QwAlarm =>)
   END_RUNG
   RUNG wire#powerrail
      Contact( "AV-79.08" )
   END_RUNG wire#w1
   RUNG wire#powerrail
      I_Contact( "AV-79.08" )
   END_RUNG wire#w2
   // the same network as SCL:
   #"AV-79.08"(LOCK := #lock,   // "Valve"
               LIOP_SEL := #Init,
               L_AUT := #Init,
               L_REMOTE := #Init,
               L_RESET := #Reset,
               FB_OPEN := "AV-79.08",
               FB_CLOSE := NOT "AV-79.08",
               L_MON := #Init,
               INSTANCE := 'AV-79.08',
               QCMD_OP => "AV-79.08");
END_REGION

REGION Network 84: AV-79.09
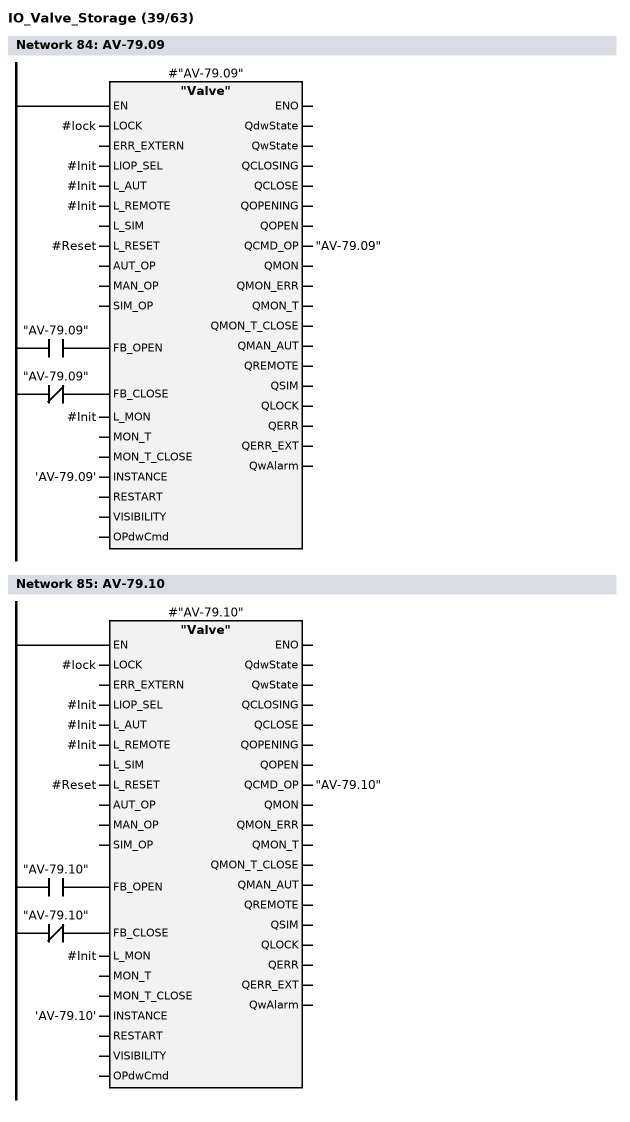
   RUNG wire#powerrail
      #"AV-79.09"(FB_OPEN := wire#w1, FB_CLOSE := wire#w2, LOCK := #lock, ERR_EXTERN :=, LIOP_SEL := #Init, L_AUT := #Init, L_REMOTE := #Init, L_SIM :=, L_RESET := #Reset, AUT_OP :=, MAN_OP :=, SIM_OP :=, L_MON := #Init, MON_T :=, MON_T_CLOSE :=, INSTANCE := 'AV-79.09', RESTART :=, VISIBILITY :=, OPdwCmd :=, QdwState =>, QwState =>, QCLOSING =>, QCLOSE =>, QOPENING =>, QOPEN =>, QCMD_OP => "AV-79.09", QMON =>, QMON_ERR =>, QMON_T =>, QMON_T_CLOSE =>, QMAN_AUT =>, QREMOTE =>, QSIM =>, QLOCK =>, QERR =>, QERR_EXT =>, QwAlarm =>)
   END_RUNG
   RUNG wire#powerrail
      Contact( "AV-79.09" )
   END_RUNG wire#w1
   RUNG wire#powerrail
      I_Contact( "AV-79.09" )
   END_RUNG wire#w2
   // the same network as SCL:
   #"AV-79.09"(LOCK := #lock,   // "Valve"
               LIOP_SEL := #Init,
               L_AUT := #Init,
               L_REMOTE := #Init,
               L_RESET := #Reset,
               FB_OPEN := "AV-79.09",
               FB_CLOSE := NOT "AV-79.09",
               L_MON := #Init,
               INSTANCE := 'AV-79.09',
               QCMD_OP => "AV-79.09");
END_REGION

REGION Network 85: AV-79.10
   RUNG wire#powerrail
      #"AV-79.10"(FB_OPEN := wire#w1, FB_CLOSE := wire#w2, LOCK := #lock, ERR_EXTERN :=, LIOP_SEL := #Init, L_AUT := #Init, L_REMOTE := #Init, L_SIM :=, L_RESET := #Reset, AUT_OP :=, MAN_OP :=, SIM_OP :=, L_MON := #Init, MON_T :=, MON_T_CLOSE :=, INSTANCE := 'AV-79.10', RESTART :=, VISIBILITY :=, OPdwCmd :=, QdwState =>, QwState =>, QCLOSING =>, QCLOSE =>, QOPENING =>, QOPEN =>, QCMD_OP => "AV-79.10", QMON =>, QMON_ERR =>, QMON_T =>, QMON_T_CLOSE =>, QMAN_AUT =>, QREMOTE =>, QSIM =>, QLOCK =>, QERR =>, QERR_EXT =>, QwAlarm =>)
   END_RUNG
   RUNG wire#powerrail
      Contact( "AV-79.10" )
   END_RUNG wire#w1
   RUNG wire#powerrail
      I_Contact( "AV-79.10" )
   END_RUNG wire#w2
   // the same network as SCL:
   #"AV-79.10"(LOCK := #lock,   // "Valve"
               LIOP_SEL := #Init,
               L_AUT := #Init,
               L_REMOTE := #Init,
               L_RESET := #Reset,
               FB_OPEN := "AV-79.10",
               FB_CLOSE := NOT "AV-79.10",
               L_MON := #Init,
               INSTANCE := 'AV-79.10',
               QCMD_OP => "AV-79.10");
END_REGION

REGION Network 86: AV-79.13
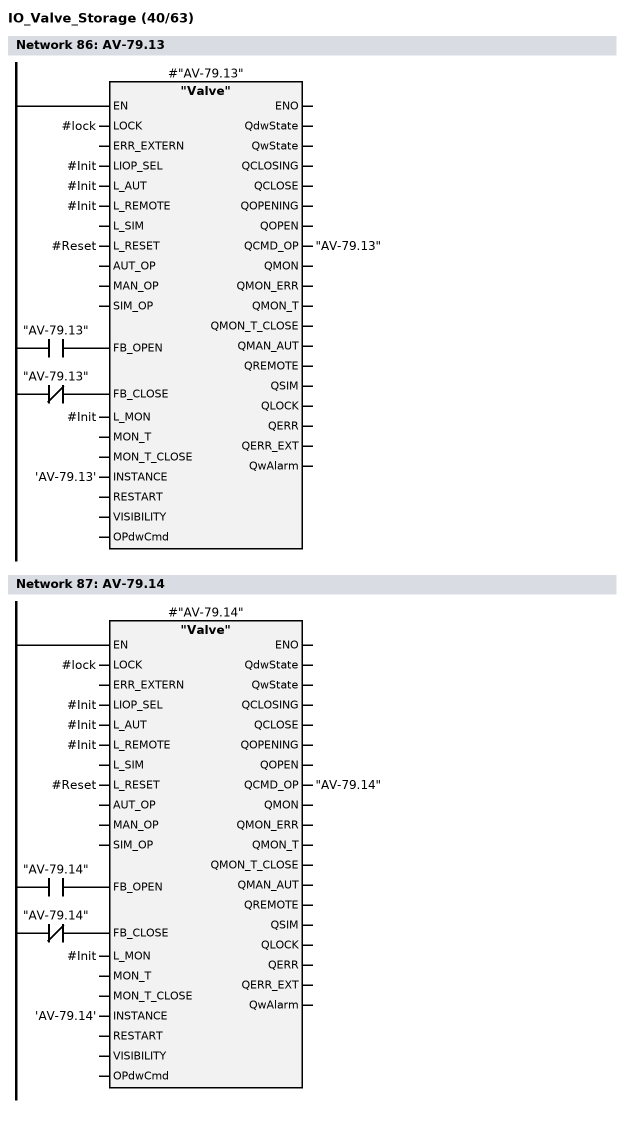
   RUNG wire#powerrail
      #"AV-79.13"(FB_OPEN := wire#w1, FB_CLOSE := wire#w2, LOCK := #lock, ERR_EXTERN :=, LIOP_SEL := #Init, L_AUT := #Init, L_REMOTE := #Init, L_SIM :=, L_RESET := #Reset, AUT_OP :=, MAN_OP :=, SIM_OP :=, L_MON := #Init, MON_T :=, MON_T_CLOSE :=, INSTANCE := 'AV-79.13', RESTART :=, VISIBILITY :=, OPdwCmd :=, QdwState =>, QwState =>, QCLOSING =>, QCLOSE =>, QOPENING =>, QOPEN =>, QCMD_OP => "AV-79.13", QMON =>, QMON_ERR =>, QMON_T =>, QMON_T_CLOSE =>, QMAN_AUT =>, QREMOTE =>, QSIM =>, QLOCK =>, QERR =>, QERR_EXT =>, QwAlarm =>)
   END_RUNG
   RUNG wire#powerrail
      Contact( "AV-79.13" )
   END_RUNG wire#w1
   RUNG wire#powerrail
      I_Contact( "AV-79.13" )
   END_RUNG wire#w2
   // the same network as SCL:
   #"AV-79.13"(LOCK := #lock,   // "Valve"
               LIOP_SEL := #Init,
               L_AUT := #Init,
               L_REMOTE := #Init,
               L_RESET := #Reset,
               FB_OPEN := "AV-79.13",
               FB_CLOSE := NOT "AV-79.13",
               L_MON := #Init,
               INSTANCE := 'AV-79.13',
               QCMD_OP => "AV-79.13");
END_REGION

REGION Network 87: AV-79.14
   RUNG wire#powerrail
      #"AV-79.14"(FB_OPEN := wire#w1, FB_CLOSE := wire#w2, LOCK := #lock, ERR_EXTERN :=, LIOP_SEL := #Init, L_AUT := #Init, L_REMOTE := #Init, L_SIM :=, L_RESET := #Reset, AUT_OP :=, MAN_OP :=, SIM_OP :=, L_MON := #Init, MON_T :=, MON_T_CLOSE :=, INSTANCE := 'AV-79.14', RESTART :=, VISIBILITY :=, OPdwCmd :=, QdwState =>, QwState =>, QCLOSING =>, QCLOSE =>, QOPENING =>, QOPEN =>, QCMD_OP => "AV-79.14", QMON =>, QMON_ERR =>, QMON_T =>, QMON_T_CLOSE =>, QMAN_AUT =>, QREMOTE =>, QSIM =>, QLOCK =>, QERR =>, QERR_EXT =>, QwAlarm =>)
   END_RUNG
   RUNG wire#powerrail
      Contact( "AV-79.14" )
   END_RUNG wire#w1
   RUNG wire#powerrail
      I_Contact( "AV-79.14" )
   END_RUNG wire#w2
   // the same network as SCL:
   #"AV-79.14"(LOCK := #lock,   // "Valve"
               LIOP_SEL := #Init,
               L_AUT := #Init,
               L_REMOTE := #Init,
               L_RESET := #Reset,
               FB_OPEN := "AV-79.14",
               FB_CLOSE := NOT "AV-79.14",
               L_MON := #Init,
               INSTANCE := 'AV-79.14',
               QCMD_OP => "AV-79.14");
END_REGION

REGION Network 88: AV-79.15
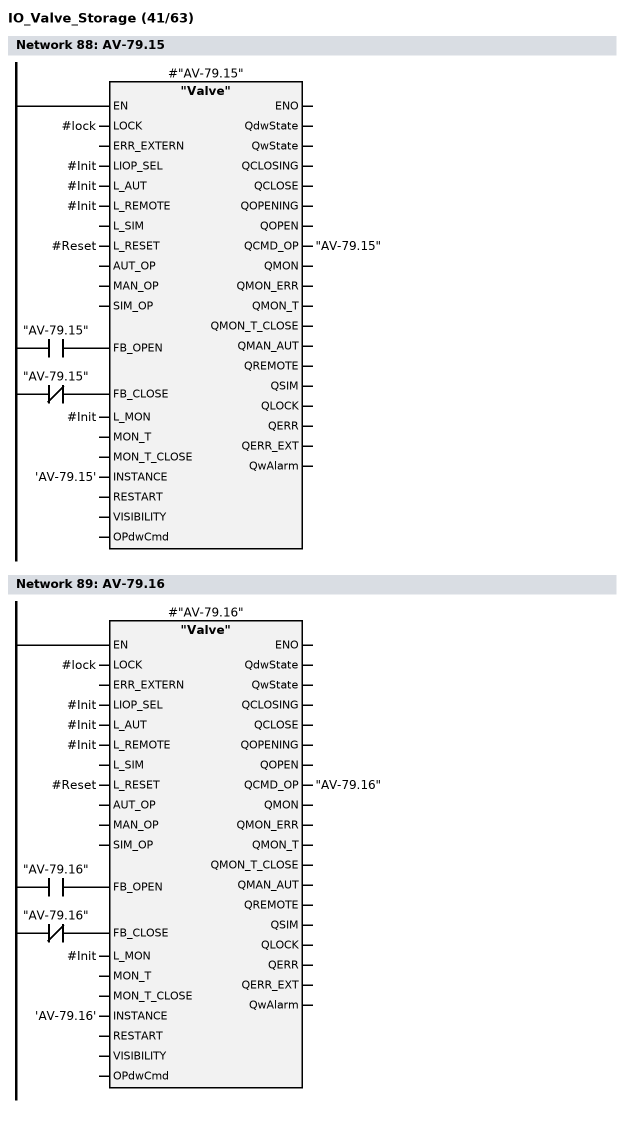
   RUNG wire#powerrail
      #"AV-79.15"(FB_OPEN := wire#w1, FB_CLOSE := wire#w2, LOCK := #lock, ERR_EXTERN :=, LIOP_SEL := #Init, L_AUT := #Init, L_REMOTE := #Init, L_SIM :=, L_RESET := #Reset, AUT_OP :=, MAN_OP :=, SIM_OP :=, L_MON := #Init, MON_T :=, MON_T_CLOSE :=, INSTANCE := 'AV-79.15', RESTART :=, VISIBILITY :=, OPdwCmd :=, QdwState =>, QwState =>, QCLOSING =>, QCLOSE =>, QOPENING =>, QOPEN =>, QCMD_OP => "AV-79.15", QMON =>, QMON_ERR =>, QMON_T =>, QMON_T_CLOSE =>, QMAN_AUT =>, QREMOTE =>, QSIM =>, QLOCK =>, QERR =>, QERR_EXT =>, QwAlarm =>)
   END_RUNG
   RUNG wire#powerrail
      Contact( "AV-79.15" )
   END_RUNG wire#w1
   RUNG wire#powerrail
      I_Contact( "AV-79.15" )
   END_RUNG wire#w2
   // the same network as SCL:
   #"AV-79.15"(LOCK := #lock,   // "Valve"
               LIOP_SEL := #Init,
               L_AUT := #Init,
               L_REMOTE := #Init,
               L_RESET := #Reset,
               FB_OPEN := "AV-79.15",
               FB_CLOSE := NOT "AV-79.15",
               L_MON := #Init,
               INSTANCE := 'AV-79.15',
               QCMD_OP => "AV-79.15");
END_REGION

REGION Network 89: AV-79.16
   RUNG wire#powerrail
      #"AV-79.16"(FB_OPEN := wire#w1, FB_CLOSE := wire#w2, LOCK := #lock, ERR_EXTERN :=, LIOP_SEL := #Init, L_AUT := #Init, L_REMOTE := #Init, L_SIM :=, L_RESET := #Reset, AUT_OP :=, MAN_OP :=, SIM_OP :=, L_MON := #Init, MON_T :=, MON_T_CLOSE :=, INSTANCE := 'AV-79.16', RESTART :=, VISIBILITY :=, OPdwCmd :=, QdwState =>, QwState =>, QCLOSING =>, QCLOSE =>, QOPENING =>, QOPEN =>, QCMD_OP => "AV-79.16", QMON =>, QMON_ERR =>, QMON_T =>, QMON_T_CLOSE =>, QMAN_AUT =>, QREMOTE =>, QSIM =>, QLOCK =>, QERR =>, QERR_EXT =>, QwAlarm =>)
   END_RUNG
   RUNG wire#powerrail
      Contact( "AV-79.16" )
   END_RUNG wire#w1
   RUNG wire#powerrail
      I_Contact( "AV-79.16" )
   END_RUNG wire#w2
   // the same network as SCL:
   #"AV-79.16"(LOCK := #lock,   // "Valve"
               LIOP_SEL := #Init,
               L_AUT := #Init,
               L_REMOTE := #Init,
               L_RESET := #Reset,
               FB_OPEN := "AV-79.16",
               FB_CLOSE := NOT "AV-79.16",
               L_MON := #Init,
               INSTANCE := 'AV-79.16',
               QCMD_OP => "AV-79.16");
END_REGION

REGION Network 90: AV-79.17
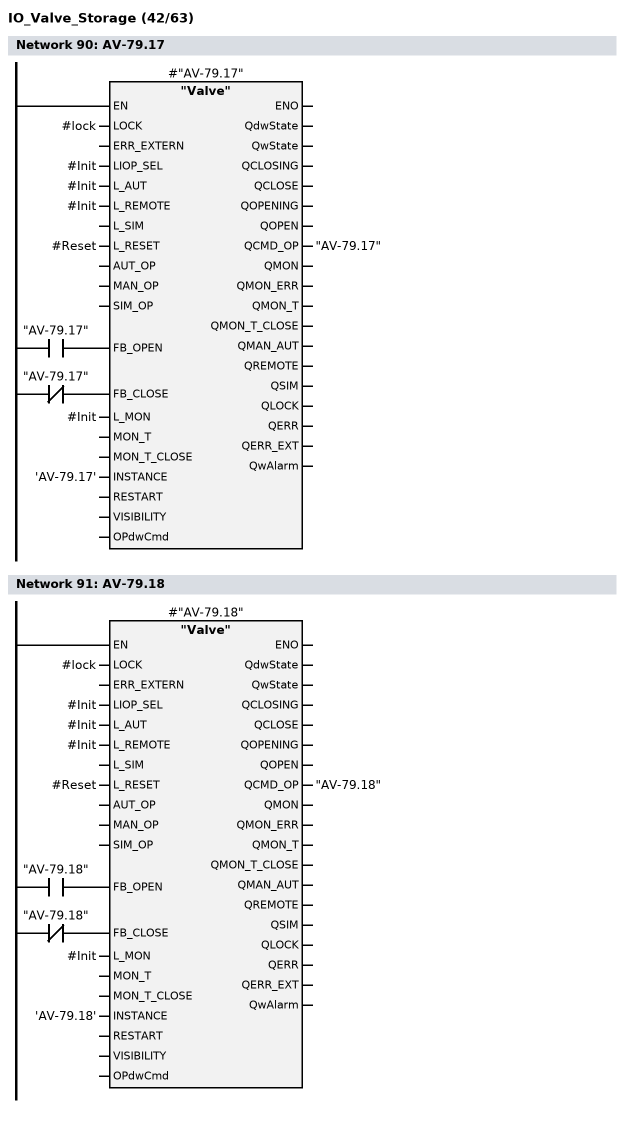
   RUNG wire#powerrail
      #"AV-79.17"(FB_OPEN := wire#w1, FB_CLOSE := wire#w2, LOCK := #lock, ERR_EXTERN :=, LIOP_SEL := #Init, L_AUT := #Init, L_REMOTE := #Init, L_SIM :=, L_RESET := #Reset, AUT_OP :=, MAN_OP :=, SIM_OP :=, L_MON := #Init, MON_T :=, MON_T_CLOSE :=, INSTANCE := 'AV-79.17', RESTART :=, VISIBILITY :=, OPdwCmd :=, QdwState =>, QwState =>, QCLOSING =>, QCLOSE =>, QOPENING =>, QOPEN =>, QCMD_OP => "AV-79.17", QMON =>, QMON_ERR =>, QMON_T =>, QMON_T_CLOSE =>, QMAN_AUT =>, QREMOTE =>, QSIM =>, QLOCK =>, QERR =>, QERR_EXT =>, QwAlarm =>)
   END_RUNG
   RUNG wire#powerrail
      Contact( "AV-79.17" )
   END_RUNG wire#w1
   RUNG wire#powerrail
      I_Contact( "AV-79.17" )
   END_RUNG wire#w2
   // the same network as SCL:
   #"AV-79.17"(LOCK := #lock,   // "Valve"
               LIOP_SEL := #Init,
               L_AUT := #Init,
               L_REMOTE := #Init,
               L_RESET := #Reset,
               FB_OPEN := "AV-79.17",
               FB_CLOSE := NOT "AV-79.17",
               L_MON := #Init,
               INSTANCE := 'AV-79.17',
               QCMD_OP => "AV-79.17");
END_REGION

REGION Network 91: AV-79.18
   RUNG wire#powerrail
      #"AV-79.18"(FB_OPEN := wire#w1, FB_CLOSE := wire#w2, LOCK := #lock, ERR_EXTERN :=, LIOP_SEL := #Init, L_AUT := #Init, L_REMOTE := #Init, L_SIM :=, L_RESET := #Reset, AUT_OP :=, MAN_OP :=, SIM_OP :=, L_MON := #Init, MON_T :=, MON_T_CLOSE :=, INSTANCE := 'AV-79.18', RESTART :=, VISIBILITY :=, OPdwCmd :=, QdwState =>, QwState =>, QCLOSING =>, QCLOSE =>, QOPENING =>, QOPEN =>, QCMD_OP => "AV-79.18", QMON =>, QMON_ERR =>, QMON_T =>, QMON_T_CLOSE =>, QMAN_AUT =>, QREMOTE =>, QSIM =>, QLOCK =>, QERR =>, QERR_EXT =>, QwAlarm =>)
   END_RUNG
   RUNG wire#powerrail
      Contact( "AV-79.18" )
   END_RUNG wire#w1
   RUNG wire#powerrail
      I_Contact( "AV-79.18" )
   END_RUNG wire#w2
   // the same network as SCL:
   #"AV-79.18"(LOCK := #lock,   // "Valve"
               LIOP_SEL := #Init,
               L_AUT := #Init,
               L_REMOTE := #Init,
               L_RESET := #Reset,
               FB_OPEN := "AV-79.18",
               FB_CLOSE := NOT "AV-79.18",
               L_MON := #Init,
               INSTANCE := 'AV-79.18',
               QCMD_OP => "AV-79.18");
END_REGION

REGION Network 92: AV-79.19
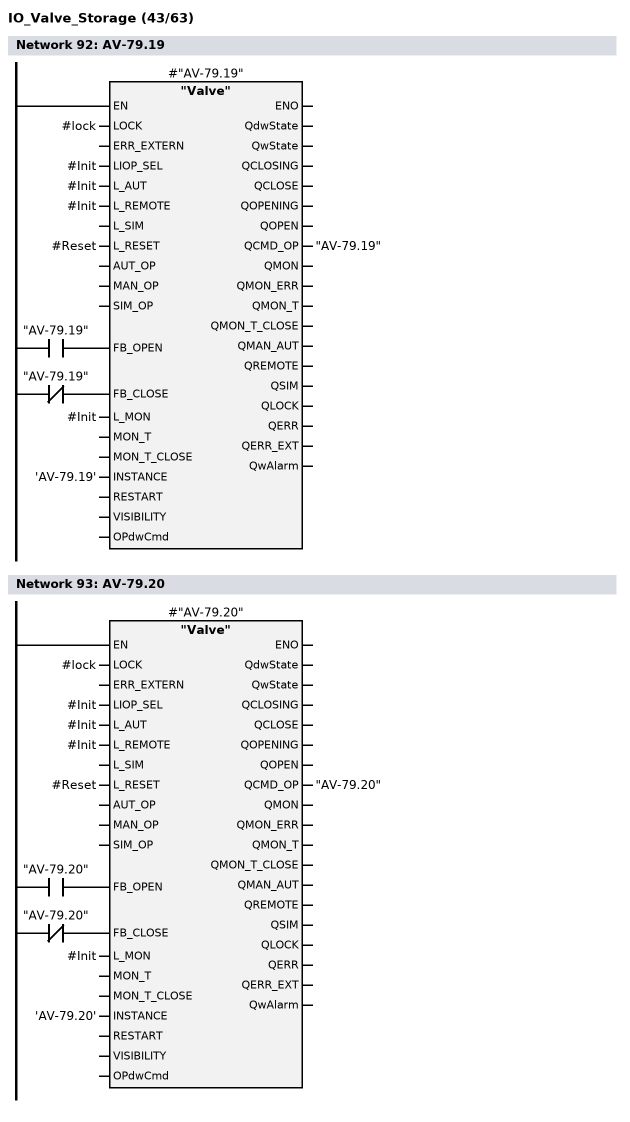
   RUNG wire#powerrail
      #"AV-79.19"(FB_OPEN := wire#w1, FB_CLOSE := wire#w2, LOCK := #lock, ERR_EXTERN :=, LIOP_SEL := #Init, L_AUT := #Init, L_REMOTE := #Init, L_SIM :=, L_RESET := #Reset, AUT_OP :=, MAN_OP :=, SIM_OP :=, L_MON := #Init, MON_T :=, MON_T_CLOSE :=, INSTANCE := 'AV-79.19', RESTART :=, VISIBILITY :=, OPdwCmd :=, QdwState =>, QwState =>, QCLOSING =>, QCLOSE =>, QOPENING =>, QOPEN =>, QCMD_OP => "AV-79.19", QMON =>, QMON_ERR =>, QMON_T =>, QMON_T_CLOSE =>, QMAN_AUT =>, QREMOTE =>, QSIM =>, QLOCK =>, QERR =>, QERR_EXT =>, QwAlarm =>)
   END_RUNG
   RUNG wire#powerrail
      Contact( "AV-79.19" )
   END_RUNG wire#w1
   RUNG wire#powerrail
      I_Contact( "AV-79.19" )
   END_RUNG wire#w2
   // the same network as SCL:
   #"AV-79.19"(LOCK := #lock,   // "Valve"
               LIOP_SEL := #Init,
               L_AUT := #Init,
               L_REMOTE := #Init,
               L_RESET := #Reset,
               FB_OPEN := "AV-79.19",
               FB_CLOSE := NOT "AV-79.19",
               L_MON := #Init,
               INSTANCE := 'AV-79.19',
               QCMD_OP => "AV-79.19");
END_REGION

REGION Network 93: AV-79.20
   RUNG wire#powerrail
      #"AV-79.20"(FB_OPEN := wire#w1, FB_CLOSE := wire#w2, LOCK := #lock, ERR_EXTERN :=, LIOP_SEL := #Init, L_AUT := #Init, L_REMOTE := #Init, L_SIM :=, L_RESET := #Reset, AUT_OP :=, MAN_OP :=, SIM_OP :=, L_MON := #Init, MON_T :=, MON_T_CLOSE :=, INSTANCE := 'AV-79.20', RESTART :=, VISIBILITY :=, OPdwCmd :=, QdwState =>, QwState =>, QCLOSING =>, QCLOSE =>, QOPENING =>, QOPEN =>, QCMD_OP => "AV-79.20", QMON =>, QMON_ERR =>, QMON_T =>, QMON_T_CLOSE =>, QMAN_AUT =>, QREMOTE =>, QSIM =>, QLOCK =>, QERR =>, QERR_EXT =>, QwAlarm =>)
   END_RUNG
   RUNG wire#powerrail
      Contact( "AV-79.20" )
   END_RUNG wire#w1
   RUNG wire#powerrail
      I_Contact( "AV-79.20" )
   END_RUNG wire#w2
   // the same network as SCL:
   #"AV-79.20"(LOCK := #lock,   // "Valve"
               LIOP_SEL := #Init,
               L_AUT := #Init,
               L_REMOTE := #Init,
               L_RESET := #Reset,
               FB_OPEN := "AV-79.20",
               FB_CLOSE := NOT "AV-79.20",
               L_MON := #Init,
               INSTANCE := 'AV-79.20',
               QCMD_OP => "AV-79.20");
END_REGION

REGION Network 94: AV-79.21
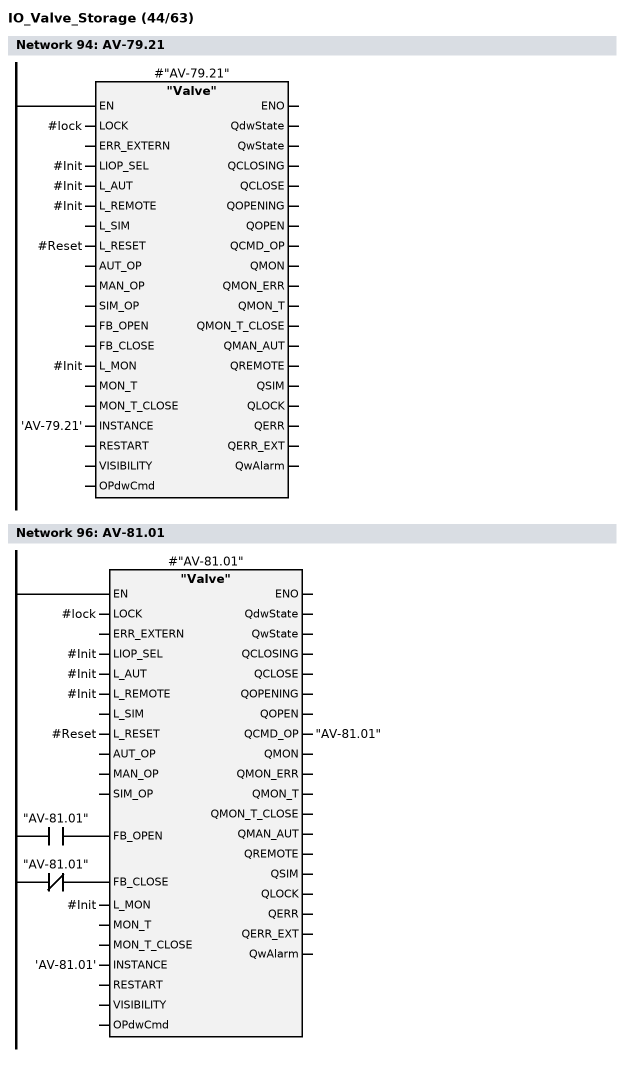
   RUNG wire#powerrail
      #"AV-79.21"(LOCK := #lock, ERR_EXTERN :=, LIOP_SEL := #Init, L_AUT := #Init, L_REMOTE := #Init, L_SIM :=, L_RESET := #Reset, AUT_OP :=, MAN_OP :=, SIM_OP :=, FB_OPEN :=, FB_CLOSE :=, L_MON := #Init, MON_T :=, MON_T_CLOSE :=, INSTANCE := 'AV-79.21', RESTART :=, VISIBILITY :=, OPdwCmd :=, QdwState =>, QwState =>, QCLOSING =>, QCLOSE =>, QOPENING =>, QOPEN =>, QCMD_OP =>, QMON =>, QMON_ERR =>, QMON_T =>, QMON_T_CLOSE =>, QMAN_AUT =>, QREMOTE =>, QSIM =>, QLOCK =>, QERR =>, QERR_EXT =>, QwAlarm =>)
   END_RUNG
   // the same network as SCL:
   #"AV-79.21"(LOCK := #lock,   // "Valve"
               LIOP_SEL := #Init,
               L_AUT := #Init,
               L_REMOTE := #Init,
               L_RESET := #Reset,
               L_MON := #Init,
               INSTANCE := 'AV-79.21');
END_REGION

REGION Network 96: AV-81.01
   RUNG wire#powerrail
      #"AV-81.01"(FB_OPEN := wire#w1, FB_CLOSE := wire#w2, LOCK := #lock, ERR_EXTERN :=, LIOP_SEL := #Init, L_AUT := #Init, L_REMOTE := #Init, L_SIM :=, L_RESET := #Reset, AUT_OP :=, MAN_OP :=, SIM_OP :=, L_MON := #Init, MON_T :=, MON_T_CLOSE :=, INSTANCE := 'AV-81.01', RESTART :=, VISIBILITY :=, OPdwCmd :=, QdwState =>, QwState =>, QCLOSING =>, QCLOSE =>, QOPENING =>, QOPEN =>, QCMD_OP => "AV-81.01", QMON =>, QMON_ERR =>, QMON_T =>, QMON_T_CLOSE =>, QMAN_AUT =>, QREMOTE =>, QSIM =>, QLOCK =>, QERR =>, QERR_EXT =>, QwAlarm =>)
   END_RUNG
   RUNG wire#powerrail
      Contact( "AV-81.01" )
   END_RUNG wire#w1
   RUNG wire#powerrail
      I_Contact( "AV-81.01" )
   END_RUNG wire#w2
   // the same network as SCL:
   #"AV-81.01"(LOCK := #lock,   // "Valve"
               LIOP_SEL := #Init,
               L_AUT := #Init,
               L_REMOTE := #Init,
               L_RESET := #Reset,
               FB_OPEN := "AV-81.01",
               FB_CLOSE := NOT "AV-81.01",
               L_MON := #Init,
               INSTANCE := 'AV-81.01',
               QCMD_OP => "AV-81.01");
END_REGION

REGION Network 97: AV-81.02
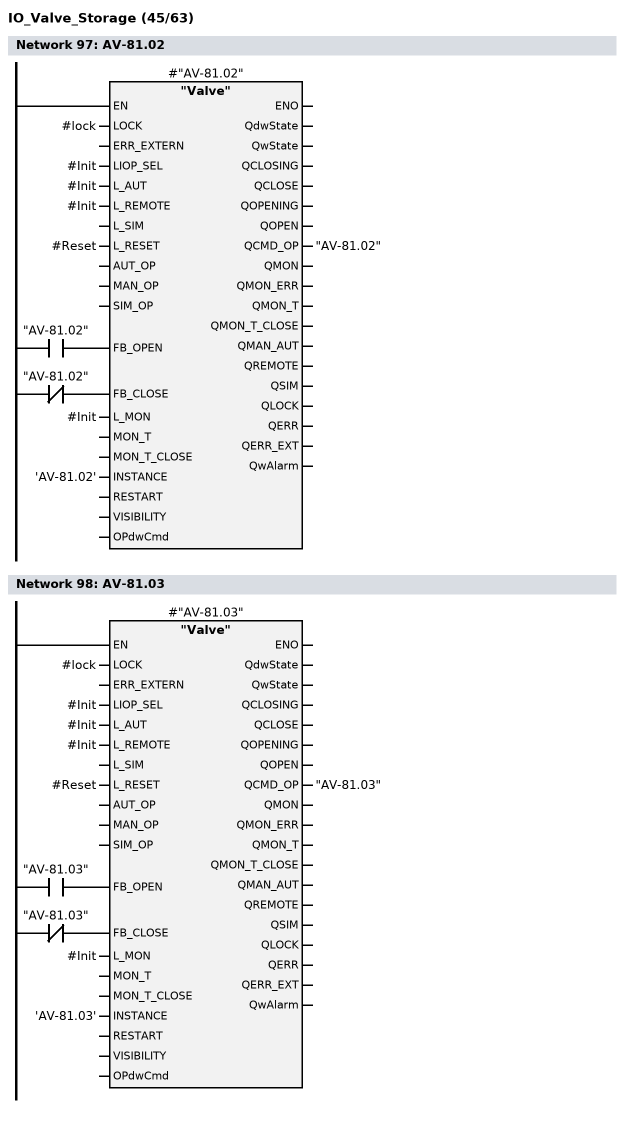
   RUNG wire#powerrail
      #"AV-81.02"(FB_OPEN := wire#w1, FB_CLOSE := wire#w2, LOCK := #lock, ERR_EXTERN :=, LIOP_SEL := #Init, L_AUT := #Init, L_REMOTE := #Init, L_SIM :=, L_RESET := #Reset, AUT_OP :=, MAN_OP :=, SIM_OP :=, L_MON := #Init, MON_T :=, MON_T_CLOSE :=, INSTANCE := 'AV-81.02', RESTART :=, VISIBILITY :=, OPdwCmd :=, QdwState =>, QwState =>, QCLOSING =>, QCLOSE =>, QOPENING =>, QOPEN =>, QCMD_OP => "AV-81.02", QMON =>, QMON_ERR =>, QMON_T =>, QMON_T_CLOSE =>, QMAN_AUT =>, QREMOTE =>, QSIM =>, QLOCK =>, QERR =>, QERR_EXT =>, QwAlarm =>)
   END_RUNG
   RUNG wire#powerrail
      Contact( "AV-81.02" )
   END_RUNG wire#w1
   RUNG wire#powerrail
      I_Contact( "AV-81.02" )
   END_RUNG wire#w2
   // the same network as SCL:
   #"AV-81.02"(LOCK := #lock,   // "Valve"
               LIOP_SEL := #Init,
               L_AUT := #Init,
               L_REMOTE := #Init,
               L_RESET := #Reset,
               FB_OPEN := "AV-81.02",
               FB_CLOSE := NOT "AV-81.02",
               L_MON := #Init,
               INSTANCE := 'AV-81.02',
               QCMD_OP => "AV-81.02");
END_REGION

REGION Network 98: AV-81.03
   RUNG wire#powerrail
      #"AV-81.03"(FB_OPEN := wire#w1, FB_CLOSE := wire#w2, LOCK := #lock, ERR_EXTERN :=, LIOP_SEL := #Init, L_AUT := #Init, L_REMOTE := #Init, L_SIM :=, L_RESET := #Reset, AUT_OP :=, MAN_OP :=, SIM_OP :=, L_MON := #Init, MON_T :=, MON_T_CLOSE :=, INSTANCE := 'AV-81.03', RESTART :=, VISIBILITY :=, OPdwCmd :=, QdwState =>, QwState =>, QCLOSING =>, QCLOSE =>, QOPENING =>, QOPEN =>, QCMD_OP => "AV-81.03", QMON =>, QMON_ERR =>, QMON_T =>, QMON_T_CLOSE =>, QMAN_AUT =>, QREMOTE =>, QSIM =>, QLOCK =>, QERR =>, QERR_EXT =>, QwAlarm =>)
   END_RUNG
   RUNG wire#powerrail
      Contact( "AV-81.03" )
   END_RUNG wire#w1
   RUNG wire#powerrail
      I_Contact( "AV-81.03" )
   END_RUNG wire#w2
   // the same network as SCL:
   #"AV-81.03"(LOCK := #lock,   // "Valve"
               LIOP_SEL := #Init,
               L_AUT := #Init,
               L_REMOTE := #Init,
               L_RESET := #Reset,
               FB_OPEN := "AV-81.03",
               FB_CLOSE := NOT "AV-81.03",
               L_MON := #Init,
               INSTANCE := 'AV-81.03',
               QCMD_OP => "AV-81.03");
END_REGION

REGION Network 99: AV-81.04
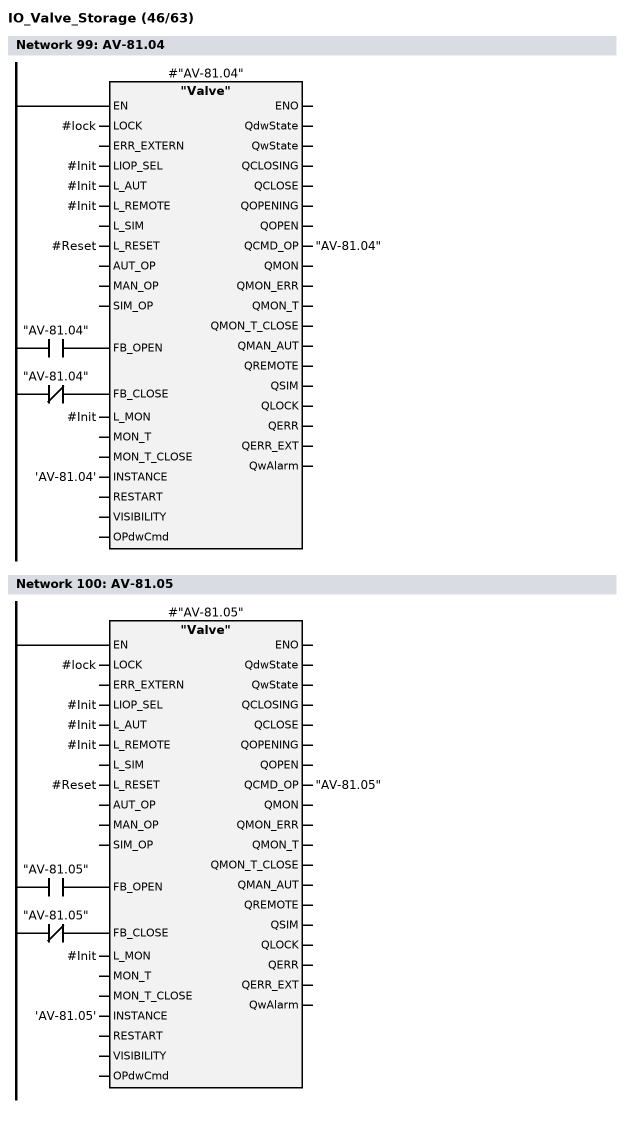
   RUNG wire#powerrail
      #"AV-81.04"(FB_OPEN := wire#w1, FB_CLOSE := wire#w2, LOCK := #lock, ERR_EXTERN :=, LIOP_SEL := #Init, L_AUT := #Init, L_REMOTE := #Init, L_SIM :=, L_RESET := #Reset, AUT_OP :=, MAN_OP :=, SIM_OP :=, L_MON := #Init, MON_T :=, MON_T_CLOSE :=, INSTANCE := 'AV-81.04', RESTART :=, VISIBILITY :=, OPdwCmd :=, QdwState =>, QwState =>, QCLOSING =>, QCLOSE =>, QOPENING =>, QOPEN =>, QCMD_OP => "AV-81.04", QMON =>, QMON_ERR =>, QMON_T =>, QMON_T_CLOSE =>, QMAN_AUT =>, QREMOTE =>, QSIM =>, QLOCK =>, QERR =>, QERR_EXT =>, QwAlarm =>)
   END_RUNG
   RUNG wire#powerrail
      Contact( "AV-81.04" )
   END_RUNG wire#w1
   RUNG wire#powerrail
      I_Contact( "AV-81.04" )
   END_RUNG wire#w2
   // the same network as SCL:
   #"AV-81.04"(LOCK := #lock,   // "Valve"
               LIOP_SEL := #Init,
               L_AUT := #Init,
               L_REMOTE := #Init,
               L_RESET := #Reset,
               FB_OPEN := "AV-81.04",
               FB_CLOSE := NOT "AV-81.04",
               L_MON := #Init,
               INSTANCE := 'AV-81.04',
               QCMD_OP => "AV-81.04");
END_REGION

REGION Network 100: AV-81.05
   RUNG wire#powerrail
      #"AV-81.05"(FB_OPEN := wire#w1, FB_CLOSE := wire#w2, LOCK := #lock, ERR_EXTERN :=, LIOP_SEL := #Init, L_AUT := #Init, L_REMOTE := #Init, L_SIM :=, L_RESET := #Reset, AUT_OP :=, MAN_OP :=, SIM_OP :=, L_MON := #Init, MON_T :=, MON_T_CLOSE :=, INSTANCE := 'AV-81.05', RESTART :=, VISIBILITY :=, OPdwCmd :=, QdwState =>, QwState =>, QCLOSING =>, QCLOSE =>, QOPENING =>, QOPEN =>, QCMD_OP => "AV-81.05", QMON =>, QMON_ERR =>, QMON_T =>, QMON_T_CLOSE =>, QMAN_AUT =>, QREMOTE =>, QSIM =>, QLOCK =>, QERR =>, QERR_EXT =>, QwAlarm =>)
   END_RUNG
   RUNG wire#powerrail
      Contact( "AV-81.05" )
   END_RUNG wire#w1
   RUNG wire#powerrail
      I_Contact( "AV-81.05" )
   END_RUNG wire#w2
   // the same network as SCL:
   #"AV-81.05"(LOCK := #lock,   // "Valve"
               LIOP_SEL := #Init,
               L_AUT := #Init,
               L_REMOTE := #Init,
               L_RESET := #Reset,
               FB_OPEN := "AV-81.05",
               FB_CLOSE := NOT "AV-81.05",
               L_MON := #Init,
               INSTANCE := 'AV-81.05',
               QCMD_OP => "AV-81.05");
END_REGION

REGION Network 101: AV-81.06
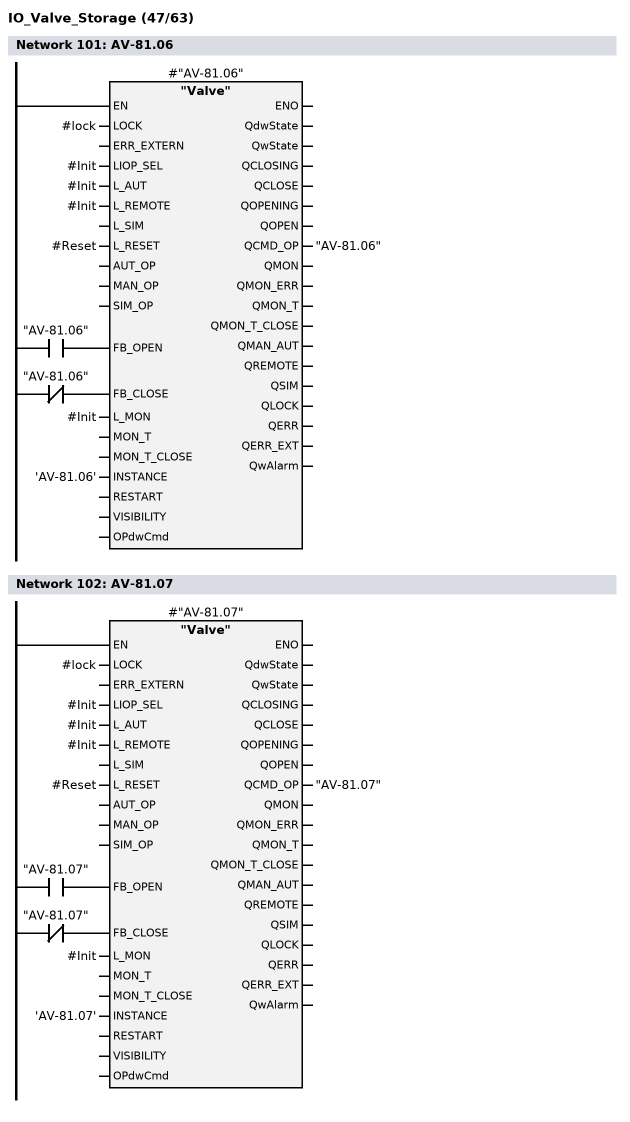
   RUNG wire#powerrail
      #"AV-81.06"(FB_OPEN := wire#w1, FB_CLOSE := wire#w2, LOCK := #lock, ERR_EXTERN :=, LIOP_SEL := #Init, L_AUT := #Init, L_REMOTE := #Init, L_SIM :=, L_RESET := #Reset, AUT_OP :=, MAN_OP :=, SIM_OP :=, L_MON := #Init, MON_T :=, MON_T_CLOSE :=, INSTANCE := 'AV-81.06', RESTART :=, VISIBILITY :=, OPdwCmd :=, QdwState =>, QwState =>, QCLOSING =>, QCLOSE =>, QOPENING =>, QOPEN =>, QCMD_OP => "AV-81.06", QMON =>, QMON_ERR =>, QMON_T =>, QMON_T_CLOSE =>, QMAN_AUT =>, QREMOTE =>, QSIM =>, QLOCK =>, QERR =>, QERR_EXT =>, QwAlarm =>)
   END_RUNG
   RUNG wire#powerrail
      Contact( "AV-81.06" )
   END_RUNG wire#w1
   RUNG wire#powerrail
      I_Contact( "AV-81.06" )
   END_RUNG wire#w2
   // the same network as SCL:
   #"AV-81.06"(LOCK := #lock,   // "Valve"
               LIOP_SEL := #Init,
               L_AUT := #Init,
               L_REMOTE := #Init,
               L_RESET := #Reset,
               FB_OPEN := "AV-81.06",
               FB_CLOSE := NOT "AV-81.06",
               L_MON := #Init,
               INSTANCE := 'AV-81.06',
               QCMD_OP => "AV-81.06");
END_REGION

REGION Network 102: AV-81.07
   RUNG wire#powerrail
      #"AV-81.07"(FB_OPEN := wire#w1, FB_CLOSE := wire#w2, LOCK := #lock, ERR_EXTERN :=, LIOP_SEL := #Init, L_AUT := #Init, L_REMOTE := #Init, L_SIM :=, L_RESET := #Reset, AUT_OP :=, MAN_OP :=, SIM_OP :=, L_MON := #Init, MON_T :=, MON_T_CLOSE :=, INSTANCE := 'AV-81.07', RESTART :=, VISIBILITY :=, OPdwCmd :=, QdwState =>, QwState =>, QCLOSING =>, QCLOSE =>, QOPENING =>, QOPEN =>, QCMD_OP => "AV-81.07", QMON =>, QMON_ERR =>, QMON_T =>, QMON_T_CLOSE =>, QMAN_AUT =>, QREMOTE =>, QSIM =>, QLOCK =>, QERR =>, QERR_EXT =>, QwAlarm =>)
   END_RUNG
   RUNG wire#powerrail
      Contact( "AV-81.07" )
   END_RUNG wire#w1
   RUNG wire#powerrail
      I_Contact( "AV-81.07" )
   END_RUNG wire#w2
   // the same network as SCL:
   #"AV-81.07"(LOCK := #lock,   // "Valve"
               LIOP_SEL := #Init,
               L_AUT := #Init,
               L_REMOTE := #Init,
               L_RESET := #Reset,
               FB_OPEN := "AV-81.07",
               FB_CLOSE := NOT "AV-81.07",
               L_MON := #Init,
               INSTANCE := 'AV-81.07',
               QCMD_OP => "AV-81.07");
END_REGION

REGION Network 103: AV-81.08
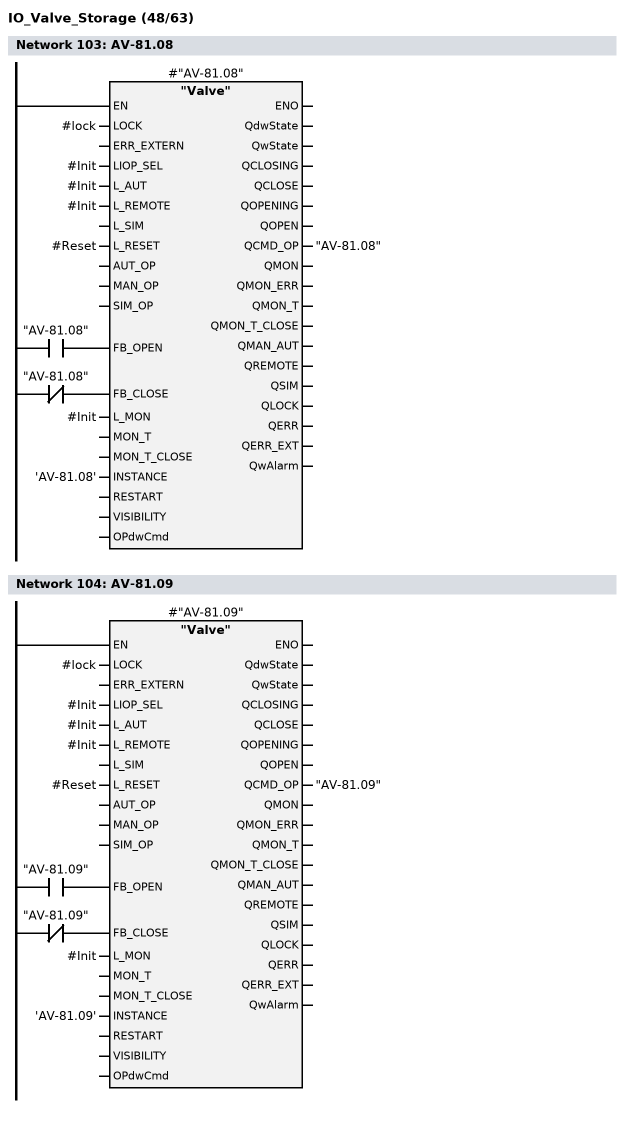
   RUNG wire#powerrail
      #"AV-81.08"(FB_OPEN := wire#w1, FB_CLOSE := wire#w2, LOCK := #lock, ERR_EXTERN :=, LIOP_SEL := #Init, L_AUT := #Init, L_REMOTE := #Init, L_SIM :=, L_RESET := #Reset, AUT_OP :=, MAN_OP :=, SIM_OP :=, L_MON := #Init, MON_T :=, MON_T_CLOSE :=, INSTANCE := 'AV-81.08', RESTART :=, VISIBILITY :=, OPdwCmd :=, QdwState =>, QwState =>, QCLOSING =>, QCLOSE =>, QOPENING =>, QOPEN =>, QCMD_OP => "AV-81.08", QMON =>, QMON_ERR =>, QMON_T =>, QMON_T_CLOSE =>, QMAN_AUT =>, QREMOTE =>, QSIM =>, QLOCK =>, QERR =>, QERR_EXT =>, QwAlarm =>)
   END_RUNG
   RUNG wire#powerrail
      Contact( "AV-81.08" )
   END_RUNG wire#w1
   RUNG wire#powerrail
      I_Contact( "AV-81.08" )
   END_RUNG wire#w2
   // the same network as SCL:
   #"AV-81.08"(LOCK := #lock,   // "Valve"
               LIOP_SEL := #Init,
               L_AUT := #Init,
               L_REMOTE := #Init,
               L_RESET := #Reset,
               FB_OPEN := "AV-81.08",
               FB_CLOSE := NOT "AV-81.08",
               L_MON := #Init,
               INSTANCE := 'AV-81.08',
               QCMD_OP => "AV-81.08");
END_REGION

REGION Network 104: AV-81.09
   RUNG wire#powerrail
      #"AV-81.09"(FB_OPEN := wire#w1, FB_CLOSE := wire#w2, LOCK := #lock, ERR_EXTERN :=, LIOP_SEL := #Init, L_AUT := #Init, L_REMOTE := #Init, L_SIM :=, L_RESET := #Reset, AUT_OP :=, MAN_OP :=, SIM_OP :=, L_MON := #Init, MON_T :=, MON_T_CLOSE :=, INSTANCE := 'AV-81.09', RESTART :=, VISIBILITY :=, OPdwCmd :=, QdwState =>, QwState =>, QCLOSING =>, QCLOSE =>, QOPENING =>, QOPEN =>, QCMD_OP => "AV-81.09", QMON =>, QMON_ERR =>, QMON_T =>, QMON_T_CLOSE =>, QMAN_AUT =>, QREMOTE =>, QSIM =>, QLOCK =>, QERR =>, QERR_EXT =>, QwAlarm =>)
   END_RUNG
   RUNG wire#powerrail
      Contact( "AV-81.09" )
   END_RUNG wire#w1
   RUNG wire#powerrail
      I_Contact( "AV-81.09" )
   END_RUNG wire#w2
   // the same network as SCL:
   #"AV-81.09"(LOCK := #lock,   // "Valve"
               LIOP_SEL := #Init,
               L_AUT := #Init,
               L_REMOTE := #Init,
               L_RESET := #Reset,
               FB_OPEN := "AV-81.09",
               FB_CLOSE := NOT "AV-81.09",
               L_MON := #Init,
               INSTANCE := 'AV-81.09',
               QCMD_OP => "AV-81.09");
END_REGION

REGION Network 105: AV-81.10
